      A     M      3.3;
      =     L      0.0;
      A     L      0.0;
      A     I    303.6;
      AN    I    303.7;
      =     M    704.4;
      A     L      0.0;
      AN    I    303.6;
      A     I    303.7;
      =     M    704.5;
NETWORK
TITLE =

      A     M      3.3;
      =     L      0.0;
      A     L      0.0;
      A     I    309.0;
      AN    I    309.1;
      AN    I    307.5;
      =     M    704.6;
      A     L      0.0;
      AN    I    309.0;
      A     I    309.1;
      A     I    307.5;
      =     M    704.7;
NETWORK
TITLE =

      A     M      3.3;
      =     L      0.0;
      A     L      0.0;
      A     I    309.2;
      AN    I    306.6;
      =     M    706.6;
      A     L      0.0;
      AN    I    309.2;
      A     I    306.6;
      =     M    706.7;
NETWORK
TITLE =
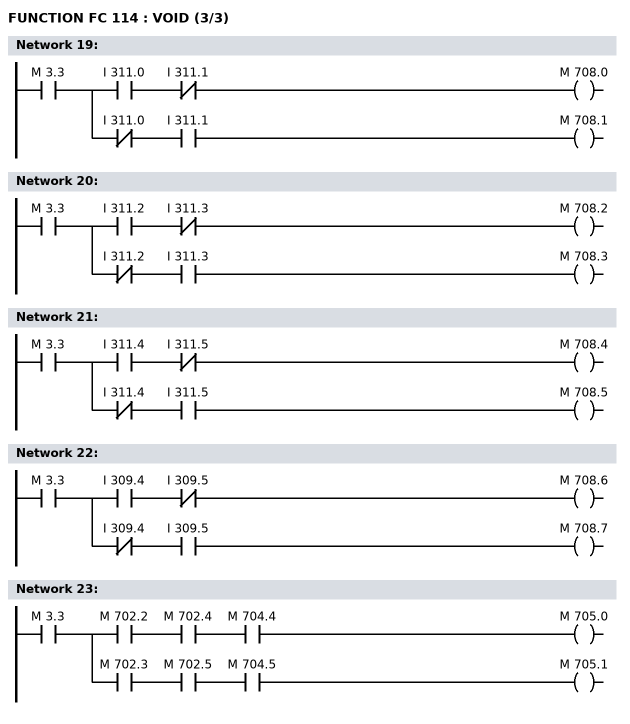

      A     M      3.3;
      =     L      0.0;
      A     L      0.0;
      A     I    311.0;
      AN    I    311.1;
      =     M    708.0;
      A     L      0.0;
      AN    I    311.0;
      A     I    311.1;
      =     M    708.1;
NETWORK
TITLE =

      A     M      3.3;
      =     L      0.0;
      A     L      0.0;
      A     I    311.2;
      AN    I    311.3;
      =     M    708.2;
      A     L      0.0;
      AN    I    311.2;
      A     I    311.3;
      =     M    708.3;
NETWORK
TITLE =

      A     M      3.3;
      =     L      0.0;
      A     L      0.0;
      A     I    311.4;
      AN    I    311.5;
      =     M    708.4;
      A     L      0.0;
      AN    I    311.4;
      A     I    311.5;
      =     M    708.5;
NETWORK
TITLE =

      A     M      3.3;
      =     L      0.0;
      A     L      0.0;
      A     I    309.4;
      AN    I    309.5;
      =     M    708.6;
      A     L      0.0;
      AN    I    309.4;
      A     I    309.5;
      =     M    708.7;
NETWORK
TITLE =

      A     M      3.3;
      =     L      0.0;
      A     L      0.0;
      A     M    702.2;
      A     M    702.4;
      A     M    704.4;
      =     M    705.0;
      A     L      0.0;
      A     M    702.3;
      A     M    702.5;
      A     M    704.5;
      =     M    705.1;
NETWORK
TITLE =

      A     M      3.3;
      =     L      0.0;
      A     L      0.0;
      A     M    702.6;
      A     M    703.0;
      A     M    703.2;
      A     M    703.4;
      A     M    703.6;
      A     M    706.6;
      =     L      0.1;
      A     L      0.1;
      BLD   102;
      =     M    705.2;
      A     L      0.1;
      A     M    704.2;
      A     M    704.6;
      =     M    705.4;
      A     L      0.0;
      A     M    702.7;
      A     M    703.1;
      A     M    703.3;
      A     M    703.5;
      A     M    703.7;
      A     M    706.7;
      =     L      0.1;
      A     L      0.1;
      BLD   102;
      =     M    705.3;
      A     L      0.1;
      A     M    704.3;
      A     M    704.7;
      =     M    705.5;
NETWORK
TITLE =
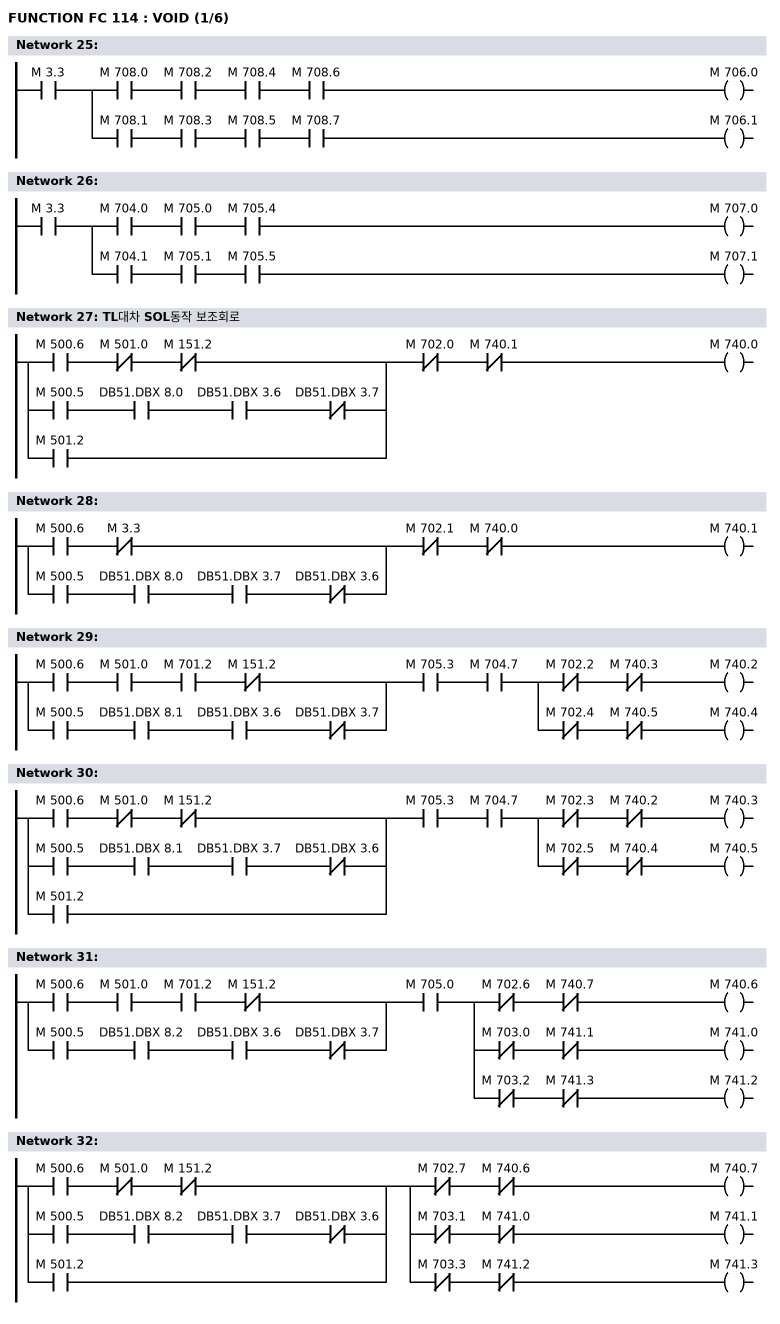

      A     M      3.3;
      =     L      0.0;
      A     L      0.0;
      A     M    708.0;
      A     M    708.2;
      A     M    708.4;
      A     M    708.6;
      =     M    706.0;
      A     L      0.0;
      A     M    708.1;
      A     M    708.3;
      A     M    708.5;
      A     M    708.7;
      =     M    706.1;
NETWORK
TITLE =

      A     M      3.3;
      =     L      0.0;
      A     L      0.0;
      A     M    704.0;
      A     M    705.0;
      A     M    705.4;
      =     M    707.0;
      A     L      0.0;
      A     M    704.1;
      A     M    705.1;
      A     M    705.5;
      =     M    707.1;
NETWORK
TITLE =TL대차 SOL동작 보조회로

      A(    ;
      A     M    500.6;
      AN    M    501.0;
      AN    M    151.2;
      O     ;
      A     M    500.5;
      A     DB51.DBX    8.0;
      A     DB51.DBX    3.6;
      AN    DB51.DBX    3.7;
      O     M    501.2;
      )     ;
      AN    M    702.0;
      AN    M    740.1;
      =     M    740.0;
NETWORK
TITLE =

      A(    ;
      A     M    500.6;
      AN    M      3.3;
      O     ;
      A     M    500.5;
      A     DB51.DBX    8.0;
      A     DB51.DBX    3.7;
      AN    DB51.DBX    3.6;
      )     ;
      AN    M    702.1;
      AN    M    740.0;
      =     M    740.1;
NETWORK
TITLE =

      A(    ;
      A     M    500.6;
      A     M    501.0;
      A     M    701.2;
      AN    M    151.2;
      O     ;
      A     M    500.5;
      A     DB51.DBX    8.1;
      A     DB51.DBX    3.6;
      AN    DB51.DBX    3.7;
      )     ;
      A     M    705.3;
      A     M    704.7;
      =     L      0.0;
      A     L      0.0;
      AN    M    702.2;
      AN    M    740.3;
      =     M    740.2;
      A     L      0.0;
      AN    M    702.4;
      AN    M    740.5;
      =     M    740.4;
NETWORK
TITLE =

      A(    ;
      A     M    500.6;
      AN    M    501.0;
      AN    M    151.2;
      O     ;
      A     M    500.5;
      A     DB51.DBX    8.1;
      A     DB51.DBX    3.7;
      AN    DB51.DBX    3.6;
      O     M    501.2;
      )     ;
      A     M    705.3;
      A     M    704.7;
      =     L      0.0;
      A     L      0.0;
      AN    M    702.3;
      AN    M    740.2;
      =     M    740.3;
      A     L      0.0;
      AN    M    702.5;
      AN    M    740.4;
      =     M    740.5;
NETWORK
TITLE =

      A(    ;
      A     M    500.6;
      A     M    501.0;
      A     M    701.2;
      AN    M    151.2;
      O     ;
      A     M    500.5;
      A     DB51.DBX    8.2;
      A     DB51.DBX    3.6;
      AN    DB51.DBX    3.7;
      )     ;
      A     M    705.0;
      =     L      0.0;
      A     L      0.0;
      AN    M    702.6;
      AN    M    740.7;
      =     M    740.6;
      A     L      0.0;
      AN    M    703.0;
      AN    M    741.1;
      =     M    741.0;
      A     L      0.0;
      AN    M    703.2;
      AN    M    741.3;
      =     M    741.2;
NETWORK
TITLE =

      A     M    500.6;
      AN    M    501.0;
      AN    M    151.2;
      O     ;
      A     M    500.5;
      A     DB51.DBX    8.2;
      A     DB51.DBX    3.7;
      AN    DB51.DBX    3.6;
      O     M    501.2;
      =     L      0.0;
      A     L      0.0;
      AN    M    702.7;
      AN    M    740.6;
      =     M    740.7;
      A     L      0.0;
      AN    M    703.1;
      AN    M    741.0;
      =     M    741.1;
      A     L      0.0;
      AN    M    703.3;
      AN    M    741.2;
      =     M    741.3;
NETWORK
TITLE =
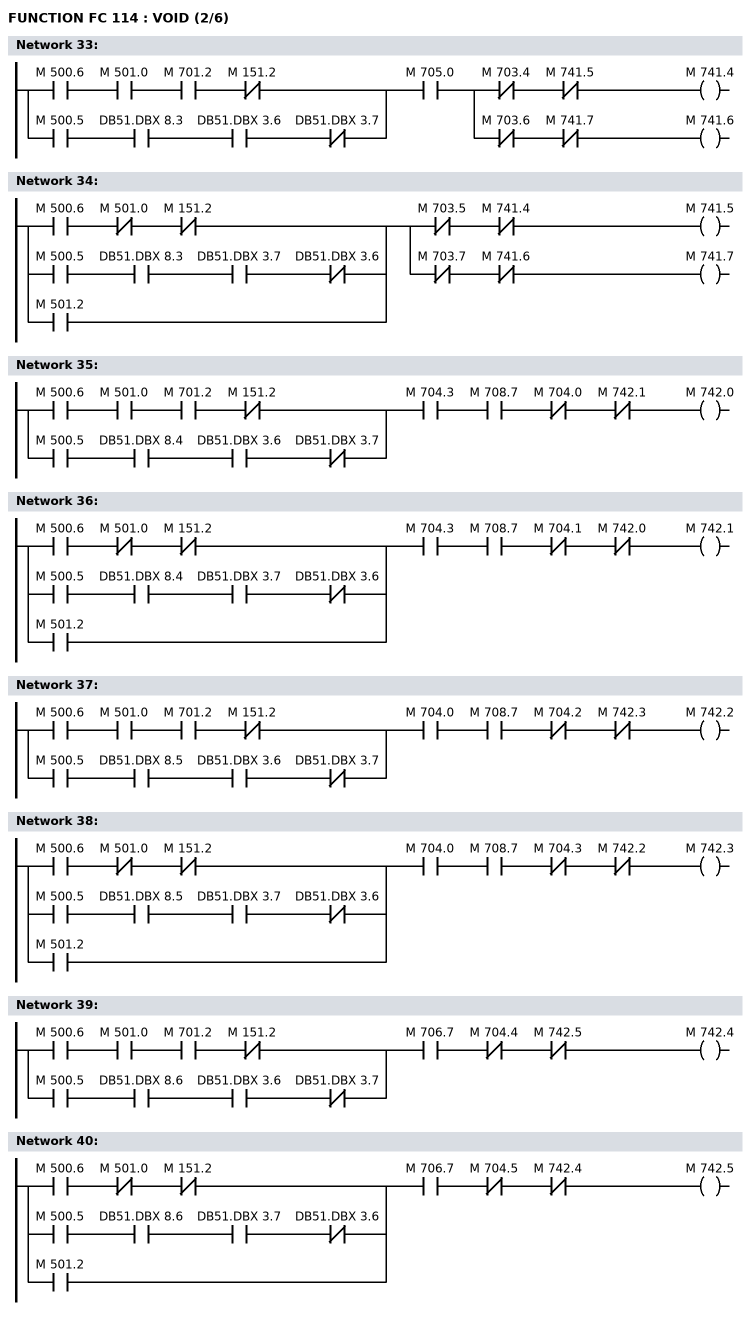

      A(    ;
      A     M    500.6;
      A     M    501.0;
      A     M    701.2;
      AN    M    151.2;
      O     ;
      A     M    500.5;
      A     DB51.DBX    8.3;
      A     DB51.DBX    3.6;
      AN    DB51.DBX    3.7;
      )     ;
      A     M    705.0;
      =     L      0.0;
      A     L      0.0;
      AN    M    703.4;
      AN    M    741.5;
      =     M    741.4;
      A     L      0.0;
      AN    M    703.6;
      AN    M    741.7;
      =     M    741.6;
NETWORK
TITLE =

      A     M    500.6;
      AN    M    501.0;
      AN    M    151.2;
      O     ;
      A     M    500.5;
      A     DB51.DBX    8.3;
      A     DB51.DBX    3.7;
      AN    DB51.DBX    3.6;
      O     M    501.2;
      =     L      0.0;
      A     L      0.0;
      AN    M    703.5;
      AN    M    741.4;
      =     M    741.5;
      A     L      0.0;
      AN    M    703.7;
      AN    M    741.6;
      =     M    741.7;
NETWORK
TITLE =

      A(    ;
      A     M    500.6;
      A     M    501.0;
      A     M    701.2;
      AN    M    151.2;
      O     ;
      A     M    500.5;
      A     DB51.DBX    8.4;
      A     DB51.DBX    3.6;
      AN    DB51.DBX    3.7;
      )     ;
      A     M    704.3;
      A     M    708.7;
      AN    M    704.0;
      AN    M    742.1;
      =     M    742.0;
NETWORK
TITLE =

      A(    ;
      A     M    500.6;
      AN    M    501.0;
      AN    M    151.2;
      O     ;
      A     M    500.5;
      A     DB51.DBX    8.4;
      A     DB51.DBX    3.7;
      AN    DB51.DBX    3.6;
      O     M    501.2;
      )     ;
      A     M    704.3;
      A     M    708.7;
      AN    M    704.1;
      AN    M    742.0;
      =     M    742.1;
NETWORK
TITLE =

      A(    ;
      A     M    500.6;
      A     M    501.0;
      A     M    701.2;
      AN    M    151.2;
      O     ;
      A     M    500.5;
      A     DB51.DBX    8.5;
      A     DB51.DBX    3.6;
      AN    DB51.DBX    3.7;
      )     ;
      A     M    704.0;
      A     M    708.7;
      AN    M    704.2;
      AN    M    742.3;
      =     M    742.2;
NETWORK
TITLE =

      A(    ;
      A     M    500.6;
      AN    M    501.0;
      AN    M    151.2;
      O     ;
      A     M    500.5;
      A     DB51.DBX    8.5;
      A     DB51.DBX    3.7;
      AN    DB51.DBX    3.6;
      O     M    501.2;
      )     ;
      A     M    704.0;
      A     M    708.7;
      AN    M    704.3;
      AN    M    742.2;
      =     M    742.3;
NETWORK
TITLE =

      A(    ;
      A     M    500.6;
      A     M    501.0;
      A     M    701.2;
      AN    M    151.2;
      O     ;
      A     M    500.5;
      A     DB51.DBX    8.6;
      A     DB51.DBX    3.6;
      AN    DB51.DBX    3.7;
      )     ;
      A     M    706.7;
      AN    M    704.4;
      AN    M    742.5;
      =     M    742.4;
NETWORK
TITLE =

      A(    ;
      A     M    500.6;
      AN    M    501.0;
      AN    M    151.2;
      O     ;
      A     M    500.5;
      A     DB51.DBX    8.6;
      A     DB51.DBX    3.7;
      AN    DB51.DBX    3.6;
      O     M    501.2;
      )     ;
      A     M    706.7;
      AN    M    704.5;
      AN    M    742.4;
      =     M    742.5;
NETWORK
TITLE =
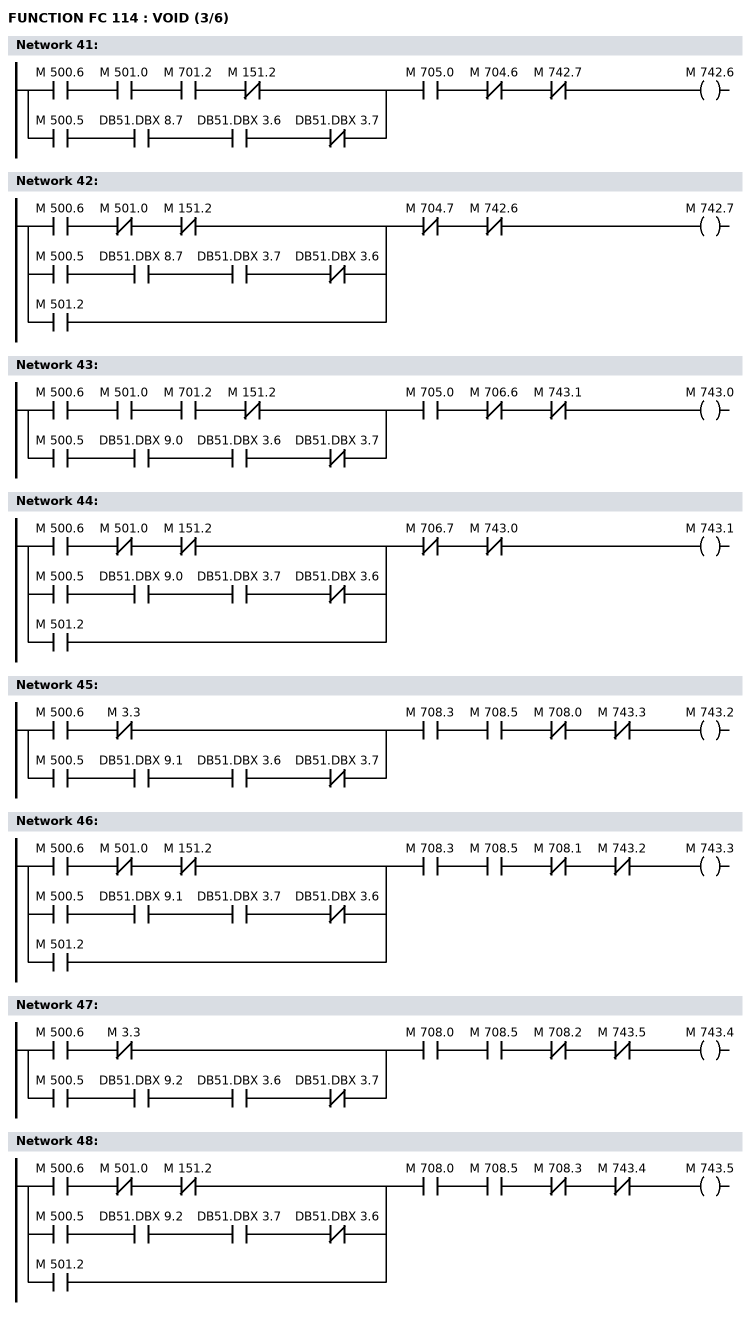

      A(    ;
      A     M    500.6;
      A     M    501.0;
      A     M    701.2;
      AN    M    151.2;
      O     ;
      A     M    500.5;
      A     DB51.DBX    8.7;
      A     DB51.DBX    3.6;
      AN    DB51.DBX    3.7;
      )     ;
      A     M    705.0;
      AN    M    704.6;
      AN    M    742.7;
      =     M    742.6;
NETWORK
TITLE =

      A(    ;
      A     M    500.6;
      AN    M    501.0;
      AN    M    151.2;
      O     ;
      A     M    500.5;
      A     DB51.DBX    8.7;
      A     DB51.DBX    3.7;
      AN    DB51.DBX    3.6;
      O     M    501.2;
      )     ;
      AN    M    704.7;
      AN    M    742.6;
      =     M    742.7;
NETWORK
TITLE =

      A(    ;
      A     M    500.6;
      A     M    501.0;
      A     M    701.2;
      AN    M    151.2;
      O     ;
      A     M    500.5;
      A     DB51.DBX    9.0;
      A     DB51.DBX    3.6;
      AN    DB51.DBX    3.7;
      )     ;
      A     M    705.0;
      AN    M    706.6;
      AN    M    743.1;
      =     M    743.0;
NETWORK
TITLE =

      A(    ;
      A     M    500.6;
      AN    M    501.0;
      AN    M    151.2;
      O     ;
      A     M    500.5;
      A     DB51.DBX    9.0;
      A     DB51.DBX    3.7;
      AN    DB51.DBX    3.6;
      O     M    501.2;
      )     ;
      AN    M    706.7;
      AN    M    743.0;
      =     M    743.1;
NETWORK
TITLE =

      A(    ;
      A     M    500.6;
      AN    M      3.3;
      O     ;
      A     M    500.5;
      A     DB51.DBX    9.1;
      A     DB51.DBX    3.6;
      AN    DB51.DBX    3.7;
      )     ;
      A     M    708.3;
      A     M    708.5;
      AN    M    708.0;
      AN    M    743.3;
      =     M    743.2;
NETWORK
TITLE =

      A(    ;
      A     M    500.6;
      AN    M    501.0;
      AN    M    151.2;
      O     ;
      A     M    500.5;
      A     DB51.DBX    9.1;
      A     DB51.DBX    3.7;
      AN    DB51.DBX    3.6;
      O     M    501.2;
      )     ;
      A     M    708.3;
      A     M    708.5;
      AN    M    708.1;
      AN    M    743.2;
      =     M    743.3;
NETWORK
TITLE =

      A(    ;
      A     M    500.6;
      AN    M      3.3;
      O     ;
      A     M    500.5;
      A     DB51.DBX    9.2;
      A     DB51.DBX    3.6;
      AN    DB51.DBX    3.7;
      )     ;
      A     M    708.0;
      A     M    708.5;
      AN    M    708.2;
      AN    M    743.5;
      =     M    743.4;
NETWORK
TITLE =

      A(    ;
      A     M    500.6;
      AN    M    501.0;
      AN    M    151.2;
      O     ;
      A     M    500.5;
      A     DB51.DBX    9.2;
      A     DB51.DBX    3.7;
      AN    DB51.DBX    3.6;
      O     M    501.2;
      )     ;
      A     M    708.0;
      A     M    708.5;
      AN    M    708.3;
      AN    M    743.4;
      =     M    743.5;
NETWORK
TITLE =
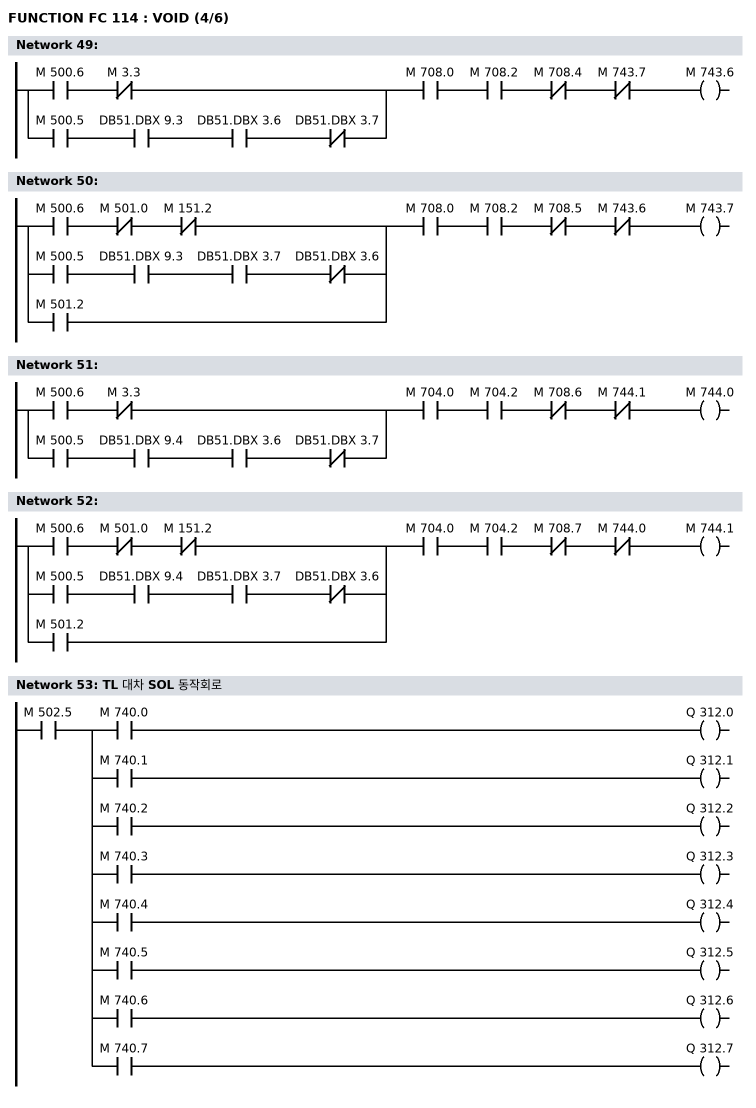

      A(    ;
      A     M    500.6;
      AN    M      3.3;
      O     ;
      A     M    500.5;
      A     DB51.DBX    9.3;
      A     DB51.DBX    3.6;
      AN    DB51.DBX    3.7;
      )     ;
      A     M    708.0;
      A     M    708.2;
      AN    M    708.4;
      AN    M    743.7;
      =     M    743.6;
NETWORK
TITLE =

      A(    ;
      A     M    500.6;
      AN    M    501.0;
      AN    M    151.2;
      O     ;
      A     M    500.5;
      A     DB51.DBX    9.3;
      A     DB51.DBX    3.7;
      AN    DB51.DBX    3.6;
      O     M    501.2;
      )     ;
      A     M    708.0;
      A     M    708.2;
      AN    M    708.5;
      AN    M    743.6;
      =     M    743.7;
NETWORK
TITLE =

      A(    ;
      A     M    500.6;
      AN    M      3.3;
      O     ;
      A     M    500.5;
      A     DB51.DBX    9.4;
      A     DB51.DBX    3.6;
      AN    DB51.DBX    3.7;
      )     ;
      A     M    704.0;
      A     M    704.2;
      AN    M    708.6;
      AN    M    744.1;
      =     M    744.0;
NETWORK
TITLE =

      A(    ;
      A     M    500.6;
      AN    M    501.0;
      AN    M    151.2;
      O     ;
      A     M    500.5;
      A     DB51.DBX    9.4;
      A     DB51.DBX    3.7;
      AN    DB51.DBX    3.6;
      O     M    501.2;
      )     ;
      A     M    704.0;
      A     M    704.2;
      AN    M    708.7;
      AN    M    744.0;
      =     M    744.1;
NETWORK
TITLE =TL 대차 SOL 동작회로

      A     M    502.5;
      =     L      0.0;
      A     L      0.0;
      A     M    740.0;
      =     Q    312.0;
      A     L      0.0;
      A     M    740.1;
      =     Q    312.1;
      A     L      0.0;
      A     M    740.2;
      =     Q    312.2;
      A     L      0.0;
      A     M    740.3;
      =     Q    312.3;
      A     L      0.0;
      A     M    740.4;
      =     Q    312.4;
      A     L      0.0;
      A     M    740.5;
      =     Q    312.5;
      A     L      0.0;
      A     M    740.6;
      =     Q    312.6;
      A     L      0.0;
      A     M    740.7;
      =     Q    312.7;
NETWORK
TITLE =
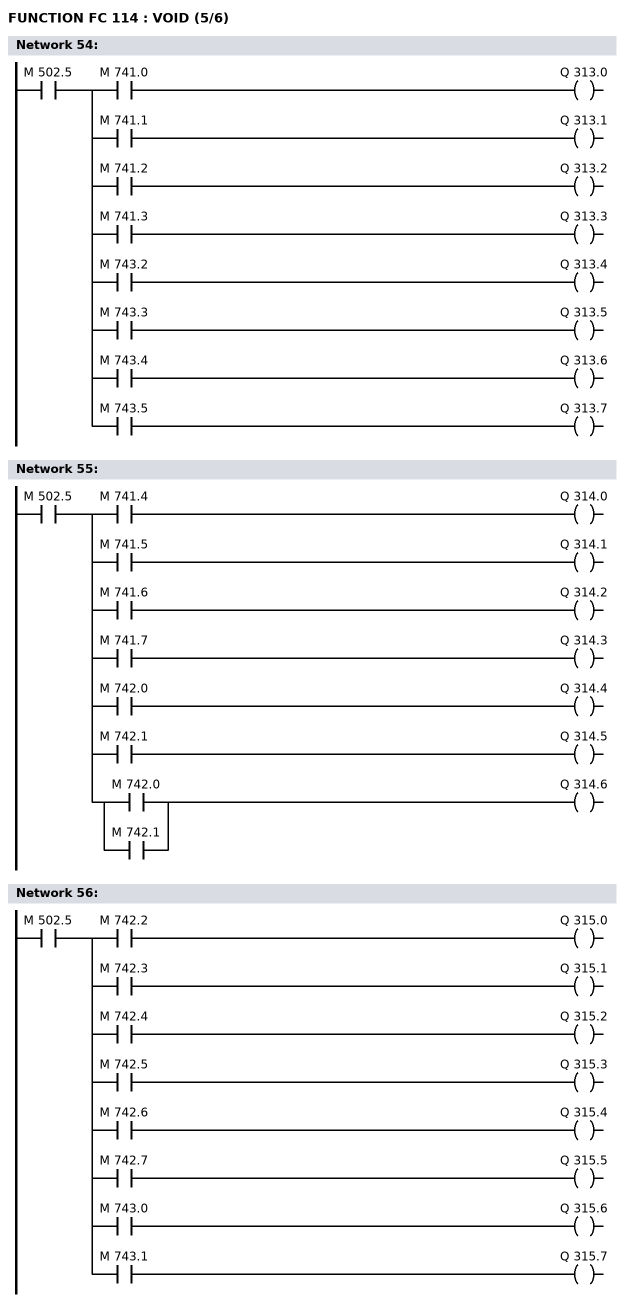

      A     M    502.5;
      =     L      0.0;
      A     L      0.0;
      A     M    741.0;
      =     Q    313.0;
      A     L      0.0;
      A     M    741.1;
      =     Q    313.1;
      A     L      0.0;
      A     M    741.2;
      =     Q    313.2;
      A     L      0.0;
      A     M    741.3;
      =     Q    313.3;
      A     L      0.0;
      A     M    743.2;
      =     Q    313.4;
      A     L      0.0;
      A     M    743.3;
      =     Q    313.5;
      A     L      0.0;
      A     M    743.4;
      =     Q    313.6;
      A     L      0.0;
      A     M    743.5;
      =     Q    313.7;
NETWORK
TITLE =

      A     M    502.5;
      =     L      0.0;
      A     L      0.0;
      A     M    741.4;
      =     Q    314.0;
      A     L      0.0;
      A     M    741.5;
      =     Q    314.1;
      A     L      0.0;
      A     M    741.6;
      =     Q    314.2;
      A     L      0.0;
      A     M    741.7;
      =     Q    314.3;
      A     L      0.0;
      A     M    742.0;
      =     Q    314.4;
      A     L      0.0;
      A     M    742.1;
      =     Q    314.5;
      A     L      0.0;
      A(    ;
      O     M    742.0;
      O     M    742.1;
      )     ;
      =     Q    314.6;
NETWORK
TITLE =

      A     M    502.5;
      =     L      0.0;
      A     L      0.0;
      A     M    742.2;
      =     Q    315.0;
      A     L      0.0;
      A     M    742.3;
      =     Q    315.1;
      A     L      0.0;
      A     M    742.4;
      =     Q    315.2;
      A     L      0.0;
      A     M    742.5;
      =     Q    315.3;
      A     L      0.0;
      A     M    742.6;
      =     Q    315.4;
      A     L      0.0;
      A     M    742.7;
      =     Q    315.5;
      A     L      0.0;
      A     M    743.0;
      =     Q    315.6;
      A     L      0.0;
      A     M    743.1;
      =     Q    315.7;
NETWORK
TITLE =
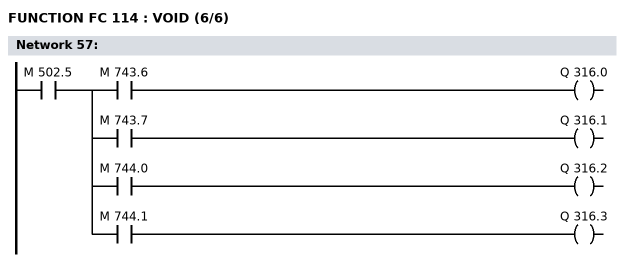

      A     M    502.5;
      =     L      0.0;
      A     L      0.0;
      A     M    743.6;
      =     Q    316.0;
      A     L      0.0;
      A     M    743.7;
      =     Q    316.1;
      A     L      0.0;
      A     M    744.0;
      =     Q    316.2;
      A     L      0.0;
      A     M    744.1;
      =     Q    316.3;
END_FUNCTION

FUNCTION FC 115 : VOID
TITLE =
VERSION : 0.1

BEGIN
NETWORK
TITLE =
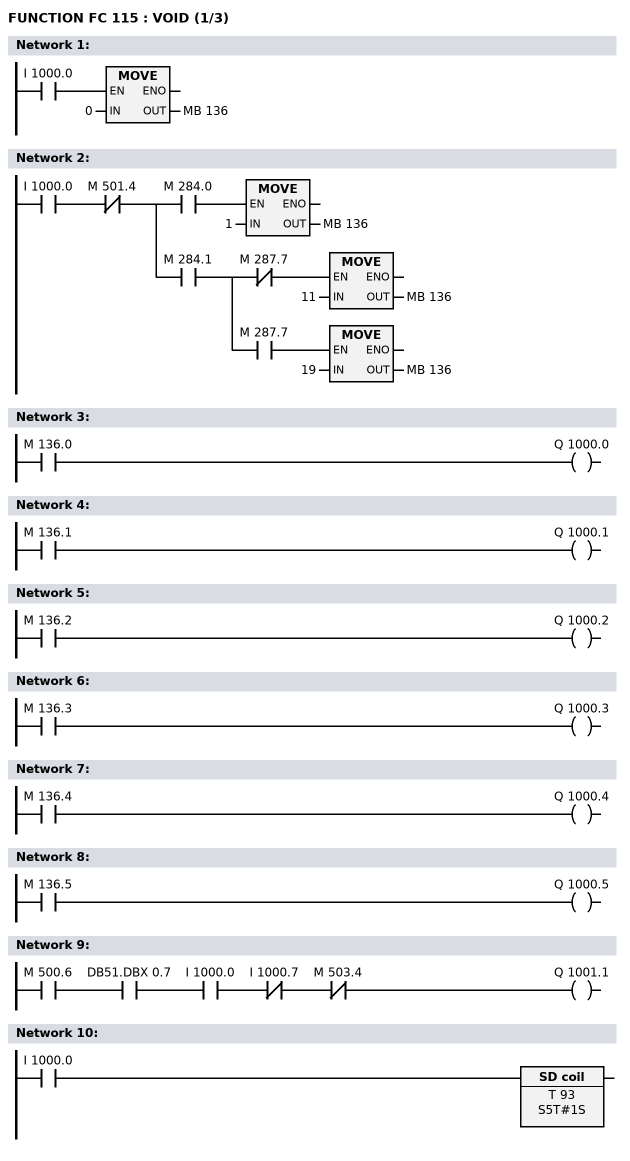

      A     I   1000.0;
      JNB   _001;
      L     0;
      T     MB   136;
_001: NOP   0;
NETWORK
TITLE =

      A     I   1000.0;
      AN    M    501.4;
      =     L      0.0;
      A     L      0.0;
      A     M    284.0;
      JNB   _002;
      L     1;
      T     MB   136;
_002: NOP   0;
      A     L      0.0;
      A     M    284.1;
      =     L      0.1;
      A     L      0.1;
      AN    M    287.7;
      JNB   _003;
      L     11;
      T     MB   136;
_003: NOP   0;
      A     L      0.1;
      A     M    287.7;
      JNB   _004;
      L     19;
      T     MB   136;
_004: NOP   0;
NETWORK
TITLE =

      A     M    136.0;
      =     Q   1000.0;
NETWORK
TITLE =

      A     M    136.1;
      =     Q   1000.1;
NETWORK
TITLE =

      A     M    136.2;
      =     Q   1000.2;
NETWORK
TITLE =

      A     M    136.3;
      =     Q   1000.3;
NETWORK
TITLE =

      A     M    136.4;
      =     Q   1000.4;
NETWORK
TITLE =

      A     M    136.5;
      =     Q   1000.5;
NETWORK
TITLE =

      A     M    500.6;
      A     DB51.DBX    0.7;
      A     I   1000.0;
      AN    I   1000.7;
      AN    M    503.4;
      =     Q   1001.1;
NETWORK
TITLE =

      A     I   1000.0;
      L     S5T#1S;
      SD    T     93;
NETWORK
TITLE =
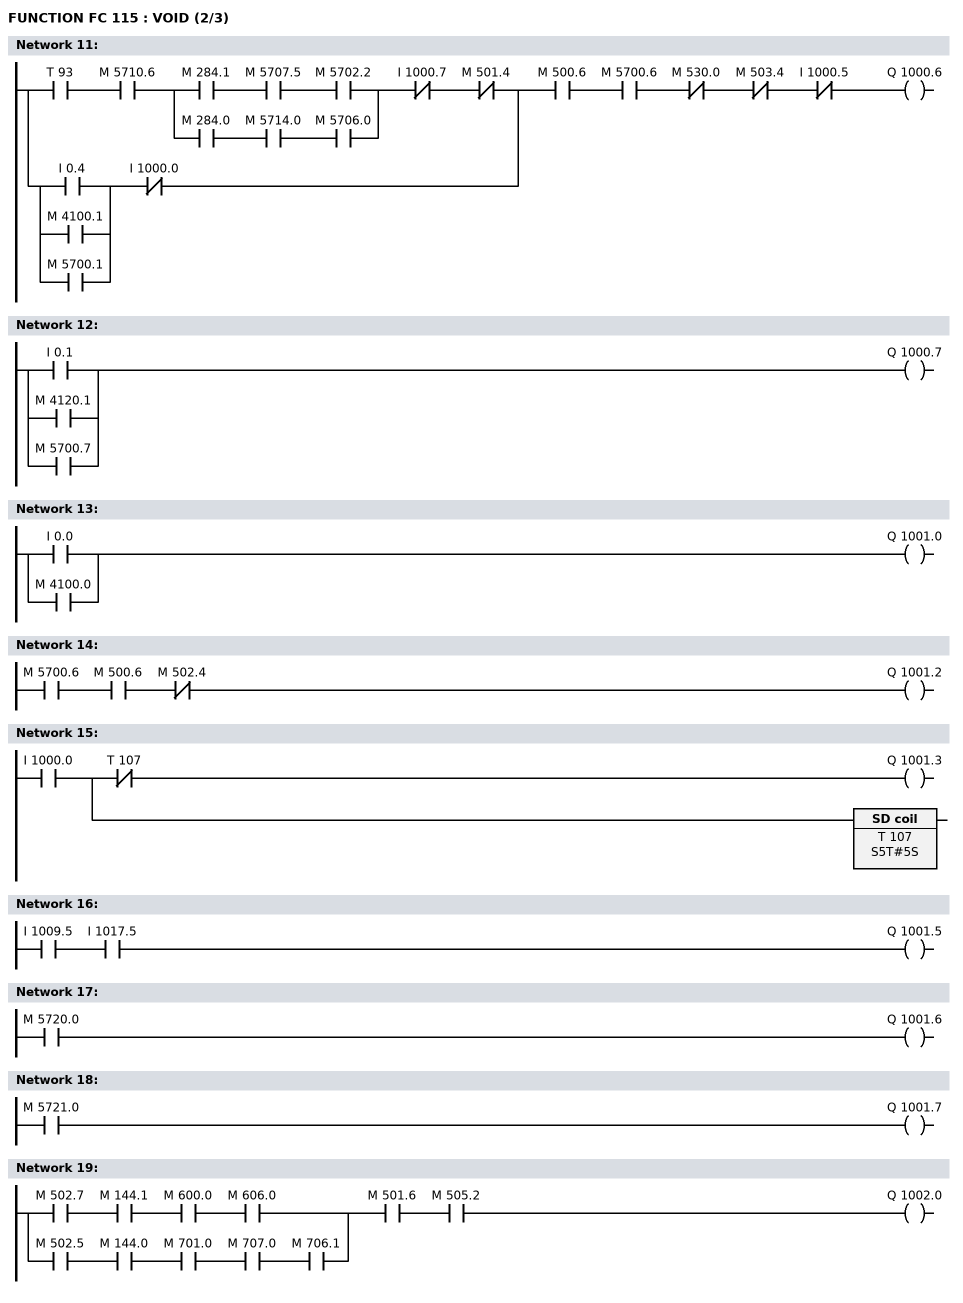

      A(    ;
      A     T     93;
      A     M   5710.6;
      A(    ;
      A     M    284.1;
      A     M   5707.5;
      A     M   5702.2;
      O     ;
      A     M    284.0;
      A     M   5714.0;
      A     M   5706.0;
      )     ;
      AN    I   1000.7;
      AN    M    501.4;
      O     ;
      A(    ;
      O     I      0.4;
      O     M   4100.1;
      O     M   5700.1;
      )     ;
      AN    I   1000.0;
      )     ;
      A     M    500.6;
      A     M   5700.6;
      AN    M    530.0;
      AN    M    503.4;
      AN    I   1000.5;
      =     Q   1000.6;
NETWORK
TITLE =

      O     I      0.1;
      O     M   4120.1;
      O     M   5700.7;
      =     Q   1000.7;
NETWORK
TITLE =

      O     I      0.0;
      O     M   4100.0;
      =     Q   1001.0;
NETWORK
TITLE =

      A     M   5700.6;
      A     M    500.6;
      AN    M    502.4;
      =     Q   1001.2;
NETWORK
TITLE =

      A     I   1000.0;
      =     L      0.0;
      A     L      0.0;
      AN    T    107;
      =     Q   1001.3;
      A     L      0.0;
      BLD   102;
      L     S5T#5S;
      SD    T    107;
NETWORK
TITLE =

      A     I   1009.5;
      A     I   1017.5;
      =     Q   1001.5;
NETWORK
TITLE =

      A     M   5720.0;
      =     Q   1001.6;
NETWORK
TITLE =

      A     M   5721.0;
      =     Q   1001.7;
NETWORK
TITLE =

      A(    ;
      A     M    502.7;
      A     M    144.1;
      A     M    600.0;
      A     M    606.0;
      O     ;
      A     M    502.5;
      A     M    144.0;
      A     M    701.0;
      A     M    707.0;
      A     M    706.1;
      )     ;
      A     M    501.6;
      A     M    505.2;
      =     Q   1002.0;
NETWORK
TITLE =
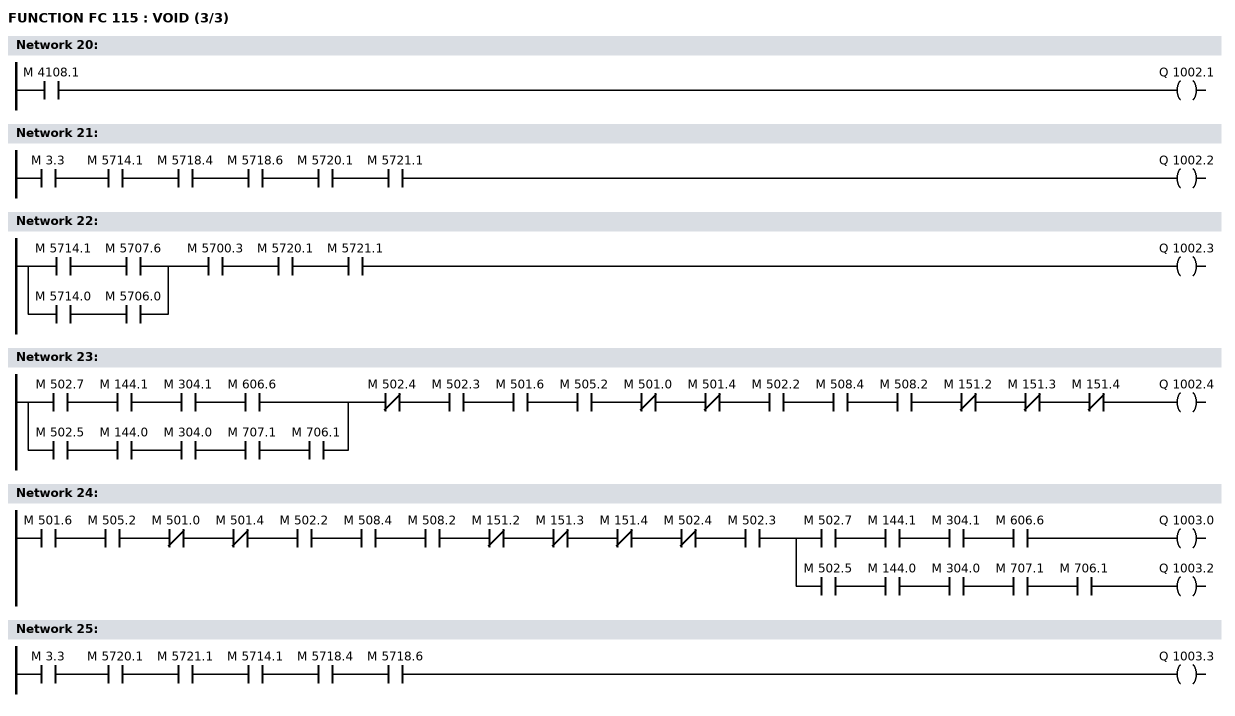

      A     M   4108.1;
      =     Q   1002.1;
NETWORK
TITLE =

      A     M      3.3;
      A     M   5714.1;
      A     M   5718.4;
      A     M   5718.6;
      A     M   5720.1;
      A     M   5721.1;
      =     Q   1002.2;
NETWORK
TITLE =

      A(    ;
      A     M   5714.1;
      A     M   5707.6;
      O     ;
      A     M   5714.0;
      A     M   5706.0;
      )     ;
      A     M   5700.3;
      A     M   5720.1;
      A     M   5721.1;
      =     Q   1002.3;
NETWORK
TITLE =

      A(    ;
      A     M    502.7;
      A     M    144.1;
      A     M    304.1;
      A     M    606.6;
      O     ;
      A     M    502.5;
      A     M    144.0;
      A     M    304.0;
      A     M    707.1;
      A     M    706.1;
      )     ;
      AN    M    502.4;
      A     M    502.3;
      A     M    501.6;
      A     M    505.2;
      AN    M    501.0;
      AN    M    501.4;
      A     M    502.2;
      A     M    508.4;
      A     M    508.2;
      AN    M    151.2;
      AN    M    151.3;
      AN    M    151.4;
      =     Q   1002.4;
NETWORK
TITLE =

      A     M    501.6;
      A     M    505.2;
      AN    M    501.0;
      AN    M    501.4;
      A     M    502.2;
      A     M    508.4;
      A     M    508.2;
      AN    M    151.2;
      AN    M    151.3;
      AN    M    151.4;
      AN    M    502.4;
      A     M    502.3;
      =     L      0.0;
      A     L      0.0;
      A     M    502.7;
      A     M    144.1;
      A     M    304.1;
      A     M    606.6;
      =     Q   1003.0;
      A     L      0.0;
      A     M    502.5;
      A     M    144.0;
      A     M    304.0;
      A     M    707.1;
      A     M    706.1;
      =     Q   1003.2;
NETWORK
TITLE =

      A     M      3.3;
      A     M   5720.1;
      A     M   5721.1;
      A     M   5714.1;
      A     M   5718.4;
      A     M   5718.6;
      =     Q   1003.3;
END_FUNCTION

FUNCTION FC 116 : VOID
TITLE =
VERSION : 0.1

BEGIN
NETWORK
TITLE =
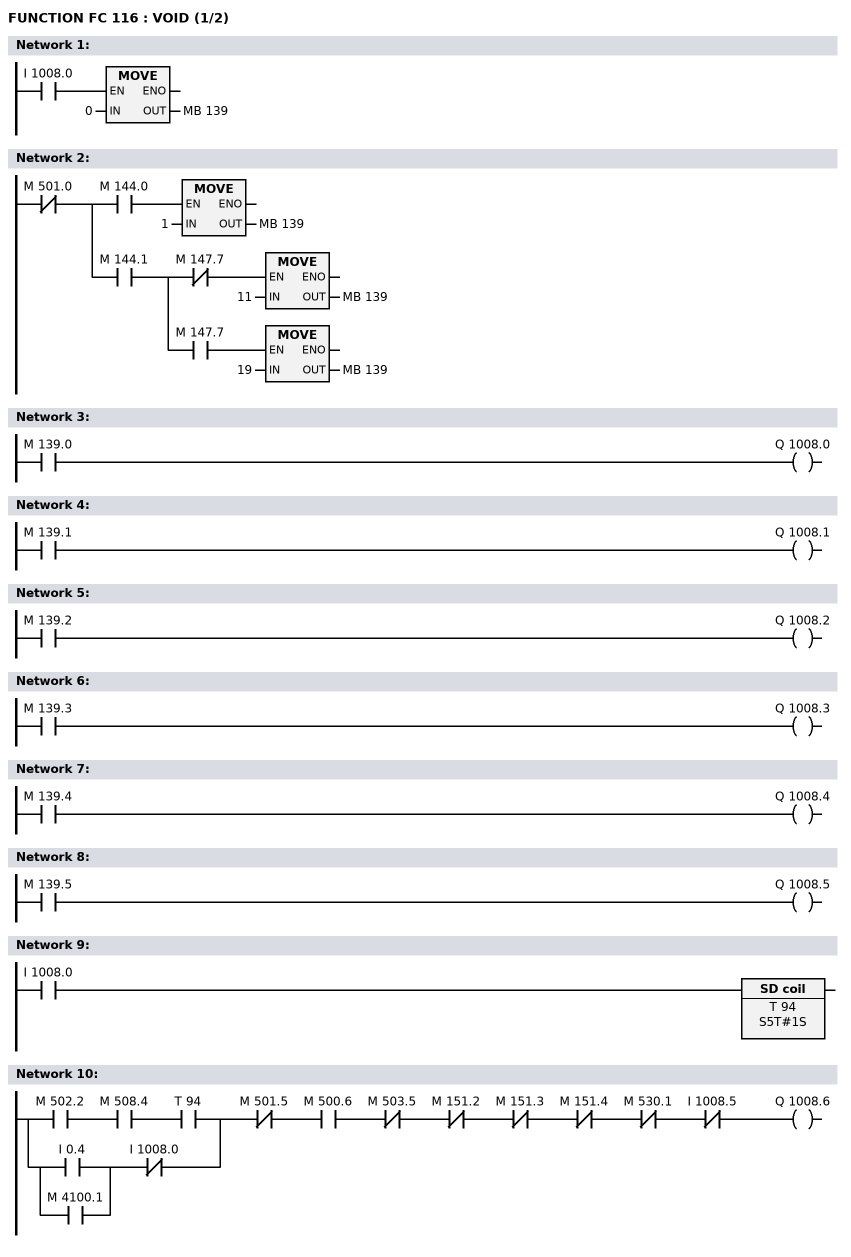

      A     I   1008.0;
      JNB   _001;
      L     0;
      T     MB   139;
_001: NOP   0;
NETWORK
TITLE =

      AN    M    501.0;
      =     L      0.0;
      A     L      0.0;
      A     M    144.0;
      JNB   _002;
      L     1;
      T     MB   139;
_002: NOP   0;
      A     L      0.0;
      A     M    144.1;
      =     L      0.1;
      A     L      0.1;
      AN    M    147.7;
      JNB   _003;
      L     11;
      T     MB   139;
_003: NOP   0;
      A     L      0.1;
      A     M    147.7;
      JNB   _004;
      L     19;
      T     MB   139;
_004: NOP   0;
NETWORK
TITLE =

      A     M    139.0;
      =     Q   1008.0;
NETWORK
TITLE =

      A     M    139.1;
      =     Q   1008.1;
NETWORK
TITLE =

      A     M    139.2;
      =     Q   1008.2;
NETWORK
TITLE =

      A     M    139.3;
      =     Q   1008.3;
NETWORK
TITLE =

      A     M    139.4;
      =     Q   1008.4;
NETWORK
TITLE =

      A     M    139.5;
      =     Q   1008.5;
NETWORK
TITLE =

      A     I   1008.0;
      L     S5T#1S;
      SD    T     94;
NETWORK
TITLE =

      A(    ;
      A     M    502.2;
      A     M    508.4;
      A     T     94;
      O     ;
      A(    ;
      O     I      0.4;
      O     M   4100.1;
      )     ;
      AN    I   1008.0;
      )     ;
      AN    M    501.5;
      A     M    500.6;
      AN    M    503.5;
      AN    M    151.2;
      AN    M    151.3;
      AN    M    151.4;
      AN    M    530.1;
      AN    I   1008.5;
      =     Q   1008.6;
NETWORK
TITLE =
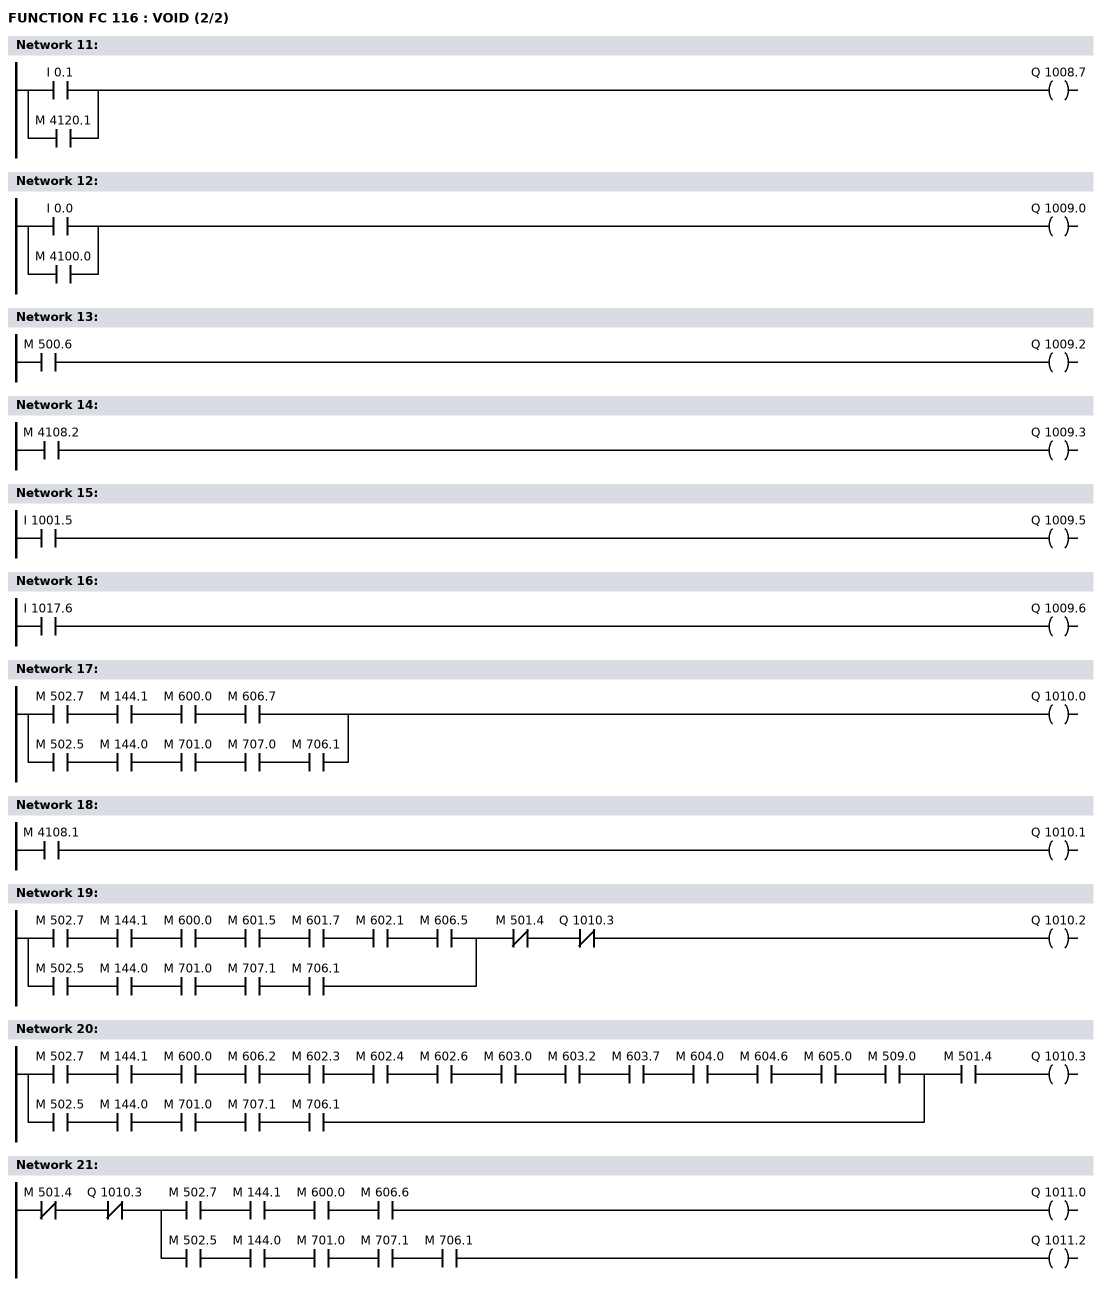

      O     I      0.1;
      O     M   4120.1;
      =     Q   1008.7;
NETWORK
TITLE =

      O     I      0.0;
      O     M   4100.0;
      =     Q   1009.0;
NETWORK
TITLE =

      A     M    500.6;
      =     Q   1009.2;
NETWORK
TITLE =

      A     M   4108.2;
      =     Q   1009.3;
NETWORK
TITLE =

      A     I   1001.5;
      =     Q   1009.5;
NETWORK
TITLE =

      A     I   1017.6;
      =     Q   1009.6;
NETWORK
TITLE =

      A     M    502.7;
      A     M    144.1;
      A     M    600.0;
      A     M    606.7;
      O     ;
      A     M    502.5;
      A     M    144.0;
      A     M    701.0;
      A     M    707.0;
      A     M    706.1;
      =     Q   1010.0;
NETWORK
TITLE =

      A     M   4108.1;
      =     Q   1010.1;
NETWORK
TITLE =

      A(    ;
      A     M    502.7;
      A     M    144.1;
      A     M    600.0;
      A     M    601.5;
      A     M    601.7;
      A     M    602.1;
      A     M    606.5;
      O     ;
      A     M    502.5;
      A     M    144.0;
      A     M    701.0;
      A     M    707.1;
      A     M    706.1;
      )     ;
      AN    M    501.4;
      AN    Q   1010.3;
      =     Q   1010.2;
NETWORK
TITLE =

      A(    ;
      A     M    502.7;
      A     M    144.1;
      A     M    600.0;
      A     M    606.2;
      A     M    602.3;
      A     M    602.4;
      A     M    602.6;
      A     M    603.0;
      A     M    603.2;
      A     M    603.7;
      A     M    604.0;
      A     M    604.6;
      A     M    605.0;
      A     M    509.0;
      O     ;
      A     M    502.5;
      A     M    144.0;
      A     M    701.0;
      A     M    707.1;
      A     M    706.1;
      )     ;
      A     M    501.4;
      =     Q   1010.3;
NETWORK
TITLE =

      AN    M    501.4;
      AN    Q   1010.3;
      =     L      0.0;
      A     L      0.0;
      A     M    502.7;
      A     M    144.1;
      A     M    600.0;
      A     M    606.6;
      =     Q   1011.0;
      A     L      0.0;
      A     M    502.5;
      A     M    144.0;
      A     M    701.0;
      A     M    707.1;
      A     M    706.1;
      =     Q   1011.2;
END_FUNCTION

FUNCTION FC 117 : VOID
TITLE =
VERSION : 0.1

BEGIN
NETWORK
TITLE =
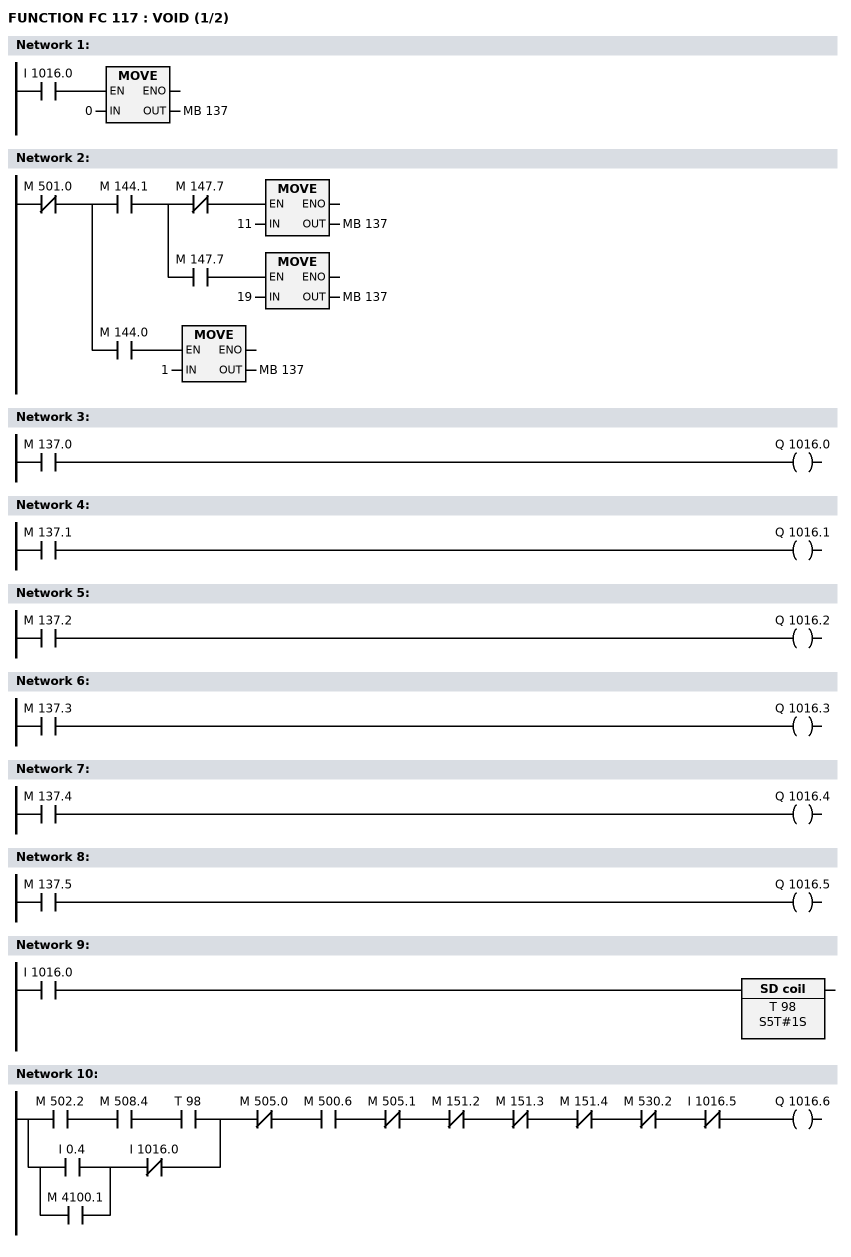

      A     I   1016.0;
      JNB   _001;
      L     0;
      T     MB   137;
_001: NOP   0;
NETWORK
TITLE =

      AN    M    501.0;
      =     L      0.0;
      A     L      0.0;
      A     M    144.1;
      =     L      0.1;
      A     L      0.1;
      AN    M    147.7;
      JNB   _002;
      L     11;
      T     MB   137;
_002: NOP   0;
      A     L      0.1;
      A     M    147.7;
      JNB   _003;
      L     19;
      T     MB   137;
_003: NOP   0;
      A     L      0.0;
      A     M    144.0;
      JNB   _004;
      L     1;
      T     MB   137;
_004: NOP   0;
NETWORK
TITLE =

      A     M    137.0;
      =     Q   1016.0;
NETWORK
TITLE =

      A     M    137.1;
      =     Q   1016.1;
NETWORK
TITLE =

      A     M    137.2;
      =     Q   1016.2;
NETWORK
TITLE =

      A     M    137.3;
      =     Q   1016.3;
NETWORK
TITLE =

      A     M    137.4;
      =     Q   1016.4;
NETWORK
TITLE =

      A     M    137.5;
      =     Q   1016.5;
NETWORK
TITLE =

      A     I   1016.0;
      L     S5T#1S;
      SD    T     98;
NETWORK
TITLE =

      A(    ;
      A     M    502.2;
      A     M    508.4;
      A     T     98;
      O     ;
      A(    ;
      O     I      0.4;
      O     M   4100.1;
      )     ;
      AN    I   1016.0;
      )     ;
      AN    M    505.0;
      A     M    500.6;
      AN    M    505.1;
      AN    M    151.2;
      AN    M    151.3;
      AN    M    151.4;
      AN    M    530.2;
      AN    I   1016.5;
      =     Q   1016.6;
NETWORK
TITLE =
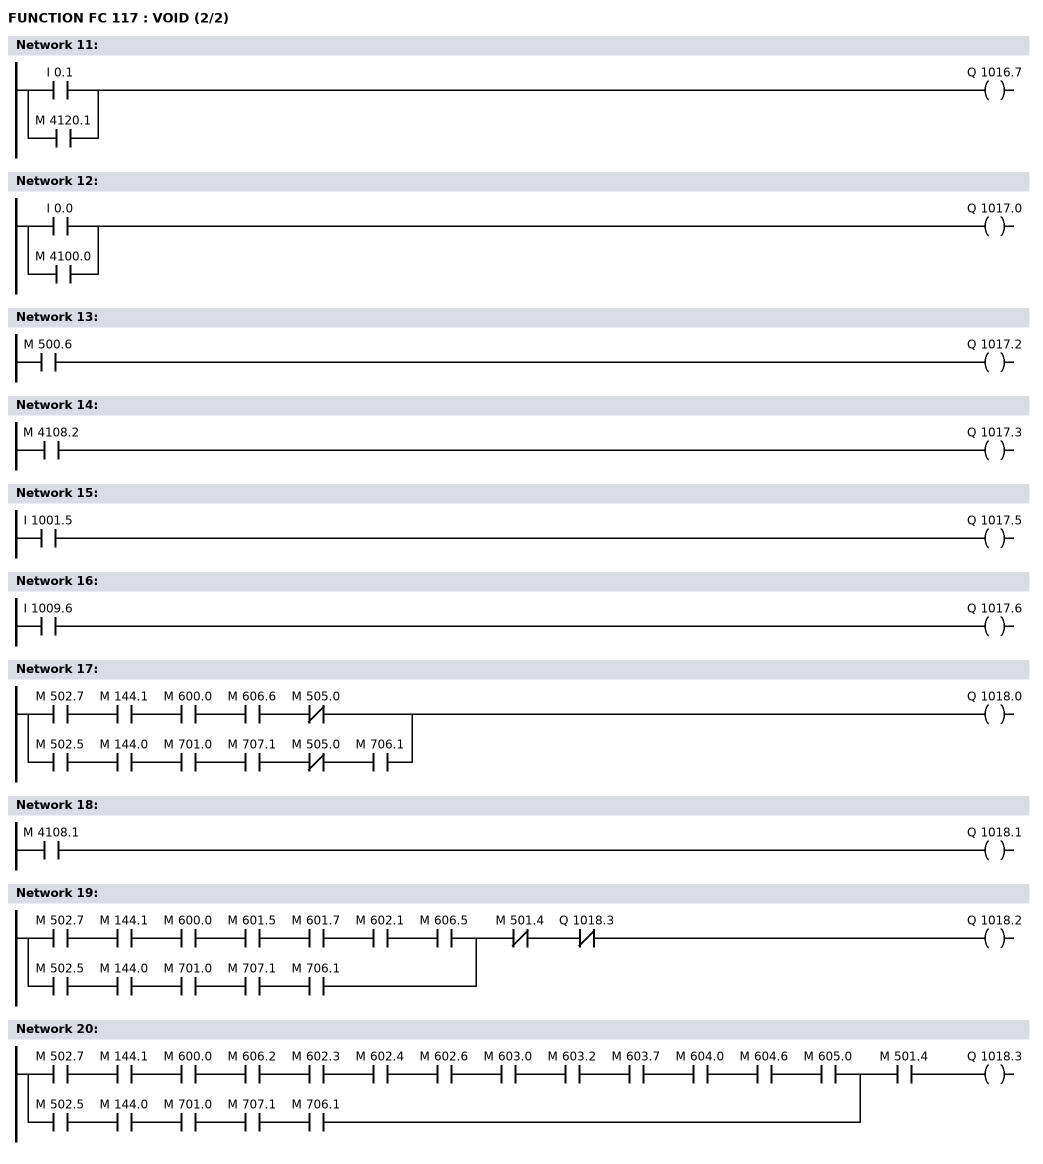

      O     I      0.1;
      O     M   4120.1;
      =     Q   1016.7;
NETWORK
TITLE =

      O     I      0.0;
      O     M   4100.0;
      =     Q   1017.0;
NETWORK
TITLE =

      A     M    500.6;
      =     Q   1017.2;
NETWORK
TITLE =

      A     M   4108.2;
      =     Q   1017.3;
NETWORK
TITLE =

      A     I   1001.5;
      =     Q   1017.5;
NETWORK
TITLE =

      A     I   1009.6;
      =     Q   1017.6;
NETWORK
TITLE =

      A     M    502.7;
      A     M    144.1;
      A     M    600.0;
      A     M    606.6;
      AN    M    505.0;
      O     ;
      A     M    502.5;
      A     M    144.0;
      A     M    701.0;
      A     M    707.1;
      AN    M    505.0;
      A     M    706.1;
      =     Q   1018.0;
NETWORK
TITLE =

      A     M   4108.1;
      =     Q   1018.1;
NETWORK
TITLE =

      A(    ;
      A     M    502.7;
      A     M    144.1;
      A     M    600.0;
      A     M    601.5;
      A     M    601.7;
      A     M    602.1;
      A     M    606.5;
      O     ;
      A     M    502.5;
      A     M    144.0;
      A     M    701.0;
      A     M    707.1;
      A     M    706.1;
      )     ;
      AN    M    501.4;
      AN    Q   1018.3;
      =     Q   1018.2;
NETWORK
TITLE =

      A(    ;
      A     M    502.7;
      A     M    144.1;
      A     M    600.0;
      A     M    606.2;
      A     M    602.3;
      A     M    602.4;
      A     M    602.6;
      A     M    603.0;
      A     M    603.2;
      A     M    603.7;
      A     M    604.0;
      A     M    604.6;
      A     M    605.0;
      O     ;
      A     M    502.5;
      A     M    144.0;
      A     M    701.0;
      A     M    707.1;
      A     M    706.1;
      )     ;
      A     M    501.4;
      =     Q   1018.3;
END_FUNCTION

FUNCTION_BLOCK FB 120
TITLE =
VERSION : 0.1


VAR
  S706_MODE : FB 402;
END_VAR
BEGIN
NETWORK
TITLE =
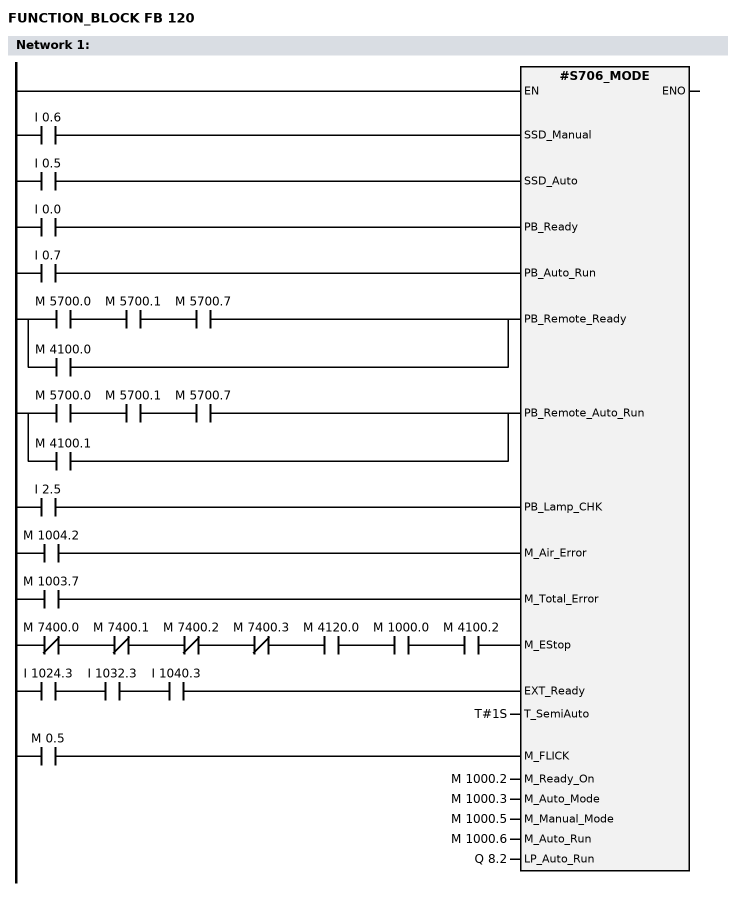

      A     I      0.6;
      =     L      0.0;
      BLD   103;
      A     I      0.5;
      =     L      0.1;
      BLD   103;
      A     I      0.0;
      =     L      0.2;
      BLD   103;
      A     I      0.7;
      =     L      0.3;
      BLD   103;
      A(    ;
      A     M   5700.0;
      A     M   5700.1;
      A     M   5700.7;
      O     M   4100.0;
      )     ;
      =     L      0.4;
      BLD   103;
      A(    ;
      A     M   5700.0;
      A     M   5700.1;
      A     M   5700.7;
      O     M   4100.1;
      )     ;
      =     L      0.5;
      BLD   103;
      A     I      2.5;
      =     L      0.6;
      BLD   103;
      A     M   1004.2;
      =     L      0.7;
      BLD   103;
      A     M   1003.7;
      =     L      1.1;
      BLD   103;
      AN    M   7400.0;
      AN    M   7400.1;
      AN    M   7400.2;
      AN    M   7400.3;
      A     M   4120.0;
      A     M   1000.0;
      A     M   4100.2;
      =     L      1.2;
      BLD   103;
      A     I   1024.3;
      A     I   1032.3;
      A     I   1040.3;
      =     L      1.3;
      BLD   103;
      A     M      0.5;
      =     L      1.5;
      BLD   103;
      CALL #S706_MODE (
           SSD_Manual               := L      0.0,
           SSD_Auto                 := L      0.1,
           PB_Ready                 := L      0.2,
           PB_Auto_Run              := L      0.3,
           PB_Remote_Ready          := L      0.4,
           PB_Remote_Auto_Run       := L      0.5,
           PB_Lamp_CHK              := L      0.6,
           M_Air_Error              := L      0.7,
           M_Total_Error            := L      1.1,
           M_EStop                  := L      1.2,
           EXT_Ready                := L      1.3,
           T_SemiAuto               := T#1S,
           M_FLICK                  := L      1.5,
           M_Ready_On               := M   1000.2,
           M_Auto_Mode              := M   1000.3,
           M_Manual_Mode            := M   1000.5,
           M_Auto_Run               := M   1000.6,
           LP_Auto_Run              := Q      8.2);
      NOP   0;
END_FUNCTION_BLOCK

DATA_BLOCK DB 120
TITLE =
VERSION : 0.0

 FB 120
BEGIN
   S706_MODE.SSD_Manual := FALSE;
   S706_MODE.SSD_Auto := TRUE;
   S706_MODE.PB_Ready := FALSE;
   S706_MODE.PB_Auto_Run := FALSE;
   S706_MODE.PB_Remote_Ready := FALSE;
   S706_MODE.PB_Remote_Auto_Run := FALSE;
   S706_MODE.PB_Lamp_CHK := FALSE;
   S706_MODE.M_Air_Error := FALSE;
   S706_MODE.M_Water_Error := FALSE;
   S706_MODE.M_Total_Error := FALSE;
   S706_MODE.M_EStop := TRUE;
   S706_MODE.EXT_Ready := TRUE;
   S706_MODE.EXT_Auto := FALSE;
   S706_MODE.T_SemiAuto := T#1S;
   S706_MODE.M_FLICK := TRUE;
   S706_MODE.M_Ready_On := TRUE;
   S706_MODE.M_Auto_Mode := TRUE;
   S706_MODE.M_SemiAuto_Mode := FALSE;
   S706_MODE.M_Manual_Mode := FALSE;
   S706_MODE.M_Auto_Run := TRUE;
   S706_MODE.LP_Ready_On := TRUE;
   S706_MODE.LP_Auto_Run := TRUE;
   S706_MODE.AUTO_MODE_DELAY.IN := FALSE;
   S706_MODE.AUTO_MODE_DELAY.PT := T#0MS;
   S706_MODE.AUTO_MODE_DELAY.Q := FALSE;
   S706_MODE.AUTO_MODE_DELAY.ET := T#0MS;
   S706_MODE.AUTO_MODE_DELAY.STATE := B#16#0;
   S706_MODE.AUTO_MODE_DELAY.STIME := T#0MS;
   S706_MODE.AUTO_MODE_DELAY.ATIME := T#0MS;
   S706_MODE.SEMI_AUTO_DELAY.IN := FALSE;
   S706_MODE.SEMI_AUTO_DELAY.PT := T#1S;
   S706_MODE.SEMI_AUTO_DELAY.Q := FALSE;
   S706_MODE.SEMI_AUTO_DELAY.ET := T#0MS;
   S706_MODE.SEMI_AUTO_DELAY.STATE := B#16#0;
   S706_MODE.SEMI_AUTO_DELAY.STIME := T#3D5H44M23S926MS;
   S706_MODE.SEMI_AUTO_DELAY.ATIME := T#3D5H44M23S950MS;
   S706_MODE.MANUAL_DELAY.IN := FALSE;
   S706_MODE.MANUAL_DELAY.PT := T#0MS;
   S706_MODE.MANUAL_DELAY.Q := FALSE;
   S706_MODE.MANUAL_DELAY.ET := T#0MS;
   S706_MODE.MANUAL_DELAY.STATE := B#16#0;
   S706_MODE.MANUAL_DELAY.STIME := T#0MS;
   S706_MODE.MANUAL_DELAY.ATIME := T#0MS;
END_DATA_BLOCK

FUNCTION FC 120 : VOID
TITLE =
VERSION : 0.1

BEGIN
NETWORK
TITLE =
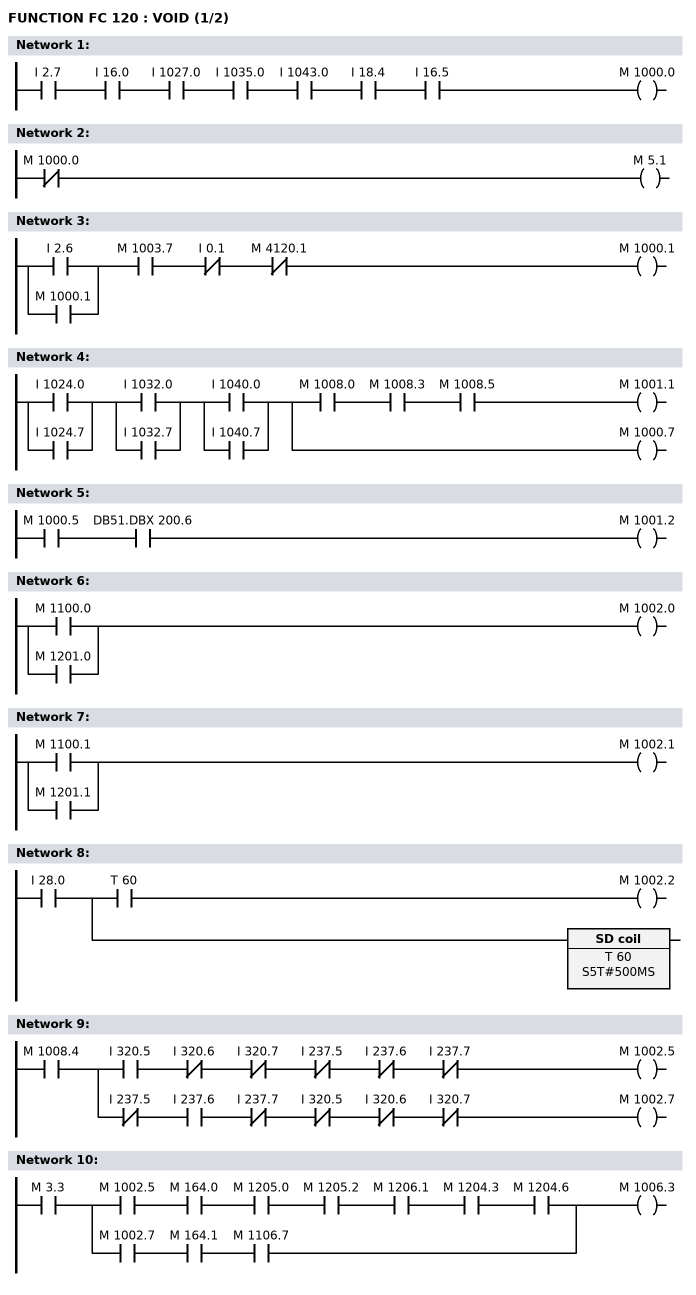

      A     I      2.7;
      A     I     16.0;
      A     I   1027.0;
      A     I   1035.0;
      A     I   1043.0;
      A     I     18.4;
      A     I     16.5;
      =     M   1000.0;
NETWORK
TITLE =

      AN    M   1000.0;
      =     M      5.1;
NETWORK
TITLE =

      A(    ;
      O     I      2.6;
      O     M   1000.1;
      )     ;
      A     M   1003.7;
      AN    I      0.1;
      AN    M   4120.1;
      =     M   1000.1;
NETWORK
TITLE =

      A(    ;
      O     I   1024.0;
      O     I   1024.7;
      )     ;
      A(    ;
      O     I   1032.0;
      O     I   1032.7;
      )     ;
      A(    ;
      O     I   1040.0;
      O     I   1040.7;
      )     ;
      =     L      0.0;
      A     L      0.0;
      A     M   1008.0;
      A     M   1008.3;
      A     M   1008.5;
      =     M   1001.1;
      A     L      0.0;
      BLD   102;
      =     M   1000.7;
NETWORK
TITLE =

      A     M   1000.5;
      A     DB51.DBX  200.6;
      =     M   1001.2;
NETWORK
TITLE =

      O     M   1100.0;
      O     M   1201.0;
      =     M   1002.0;
NETWORK
TITLE =

      O     M   1100.1;
      O     M   1201.1;
      =     M   1002.1;
NETWORK
TITLE =

      A     I     28.0;
      =     L      0.0;
      A     L      0.0;
      A     T     60;
      =     M   1002.2;
      A     L      0.0;
      BLD   102;
      L     S5T#500MS;
      SD    T     60;
NETWORK
TITLE =

      A     M   1008.4;
      =     L      0.0;
      A     L      0.0;
      A     I    320.5;
      AN    I    320.6;
      AN    I    320.7;
      AN    I    237.5;
      AN    I    237.6;
      AN    I    237.7;
      =     M   1002.5;
      A     L      0.0;
      AN    I    237.5;
      A     I    237.6;
      AN    I    237.7;
      AN    I    320.5;
      AN    I    320.6;
      AN    I    320.7;
      =     M   1002.7;
NETWORK
TITLE =

      A     M      3.3;
      A(    ;
      A     M   1002.5;
      A     M    164.0;
      A     M   1205.0;
      A     M   1205.2;
      A     M   1206.1;
      A     M   1204.3;
      A     M   1204.6;
      O     ;
      A     M   1002.7;
      A     M    164.1;
      A     M   1106.7;
      )     ;
      =     M   1006.3;
NETWORK
TITLE =
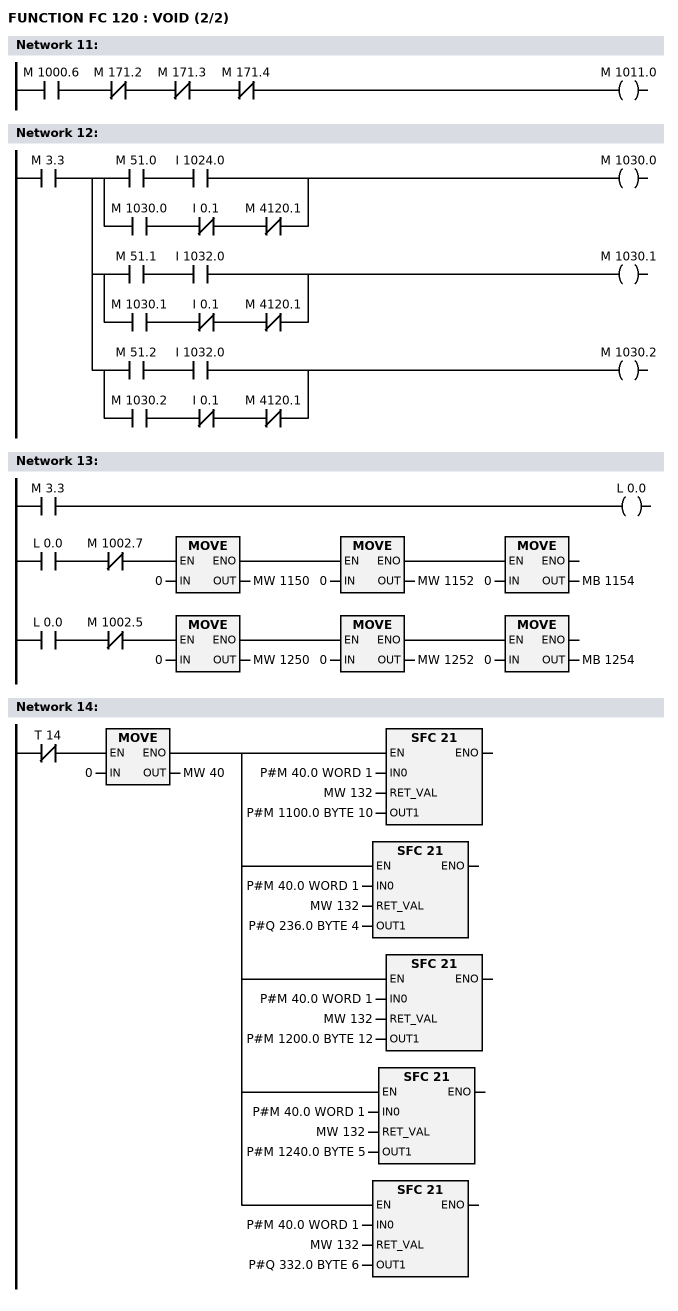

      A     M   1000.6;
      AN    M    171.2;
      AN    M    171.3;
      AN    M    171.4;
      =     M   1011.0;
NETWORK
TITLE =

      A     M      3.3;
      =     L      0.0;
      A     L      0.0;
      A(    ;
      A     M     51.0;
      A     I   1024.0;
      O     ;
      A     M   1030.0;
      AN    I      0.1;
      AN    M   4120.1;
      )     ;
      =     M   1030.0;
      A     L      0.0;
      A(    ;
      A     M     51.1;
      A     I   1032.0;
      O     ;
      A     M   1030.1;
      AN    I      0.1;
      AN    M   4120.1;
      )     ;
      =     M   1030.1;
      A     L      0.0;
      A(    ;
      A     M     51.2;
      A     I   1032.0;
      O     ;
      A     M   1030.2;
      AN    I      0.1;
      AN    M   4120.1;
      )     ;
      =     M   1030.2;
NETWORK
TITLE =

      A     M      3.3;
      =     L      0.0;
      A(    ;
      A(    ;
      A     L      0.0;
      AN    M   1002.7;
      JNB   _001;
      L     0;
      T     MW  1150;
      SET   ;
      SAVE  ;
      CLR   ;
_001: A     BR;
      )     ;
      JNB   _002;
      L     0;
      T     MW  1152;
      SET   ;
      SAVE  ;
      CLR   ;
_002: A     BR;
      )     ;
      JNB   _003;
      L     0;
      T     MB  1154;
_003: NOP   0;
      A(    ;
      A(    ;
      A     L      0.0;
      AN    M   1002.5;
      JNB   _004;
      L     0;
      T     MW  1250;
      SET   ;
      SAVE  ;
      CLR   ;
_004: A     BR;
      )     ;
      JNB   _005;
      L     0;
      T     MW  1252;
      SET   ;
      SAVE  ;
      CLR   ;
_005: A     BR;
      )     ;
      JNB   _006;
      L     0;
      T     MB  1254;
_006: NOP   0;
NETWORK
TITLE =

      AN    T     14;
      JNB   _007;
      L     0;
      T     MW    40;
      SET   ;
      SAVE  ;
      CLR   ;
_007: A     BR;
      =     L      0.0;
      A     L      0.0;
      JNB   _008;
      CALL SFC   21 (
           IN0                      := P#M 40.0 WORD 1,
           RET_VAL                  := MW   132,
           OUT1                     := P#M 1100.0 BYTE 10);
_008: NOP   0;
      A     L      0.0;
      JNB   _009;
      CALL SFC   21 (
           IN0                      := P#M 40.0 WORD 1,
           RET_VAL                  := MW   132,
           OUT1                     := P#Q 236.0 BYTE 4);
_009: NOP   0;
      A     L      0.0;
      JNB   _00a;
      CALL SFC   21 (
           IN0                      := P#M 40.0 WORD 1,
           RET_VAL                  := MW   132,
           OUT1                     := P#M 1200.0 BYTE 12);
_00a: NOP   0;
      A     L      0.0;
      JNB   _00b;
      CALL SFC   21 (
           IN0                      := P#M 40.0 WORD 1,
           RET_VAL                  := MW   132,
           OUT1                     := P#M 1240.0 BYTE 5);
_00b: NOP   0;
      A     L      0.0;
      JNB   _00c;
      CALL SFC   21 (
           IN0                      := P#M 40.0 WORD 1,
           RET_VAL                  := MW   132,
           OUT1                     := P#Q 332.0 BYTE 6);
_00c: NOP   0;
END_FUNCTION

FUNCTION_BLOCK FB 121
TITLE =
VERSION : 0.1


VAR
  S706_HOOK_PIN : FB 424;
  S706_DC_LOCK : FB 424;
  S706_ELE : FB 424;
  S706_AIR_ELE : FB 424;
END_VAR
BEGIN
NETWORK
TITLE =
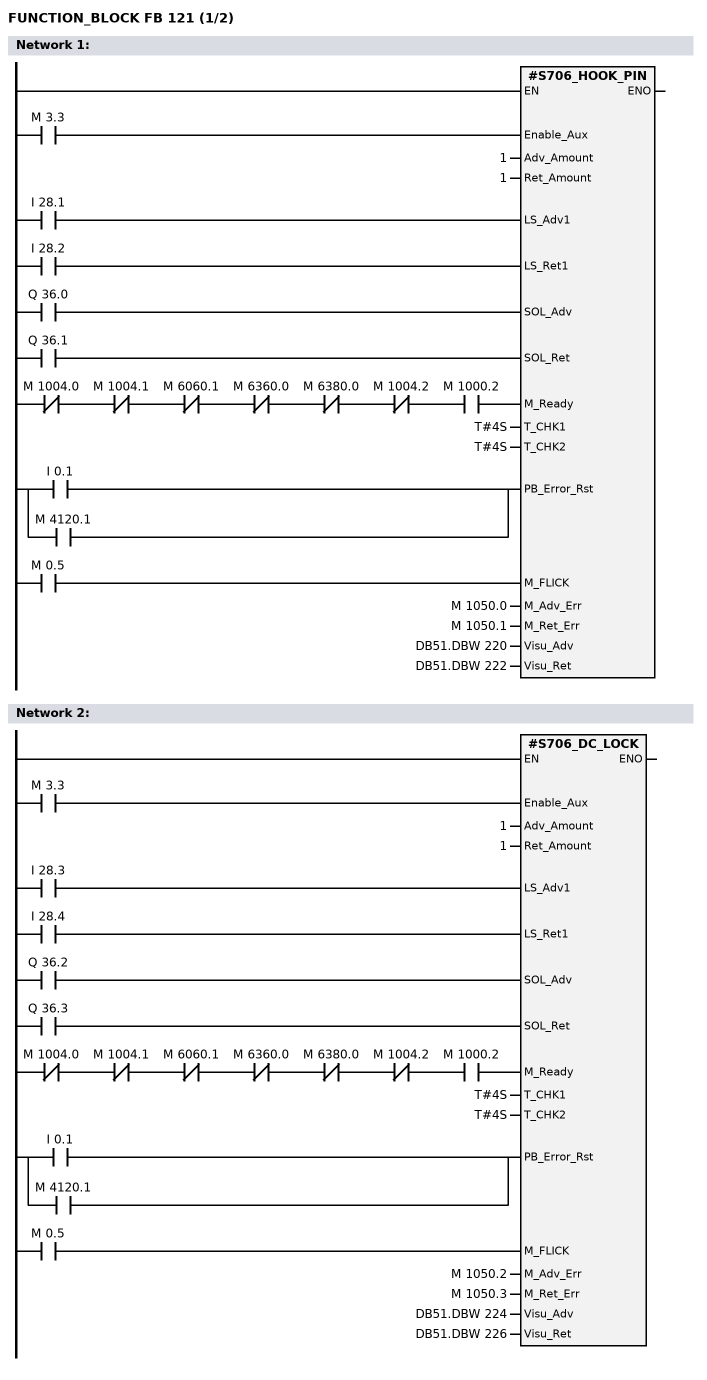

      A     M      3.3;
      =     L      0.0;
      BLD   103;
      A     I     28.1;
      =     L      0.1;
      BLD   103;
      A     I     28.2;
      =     L      0.2;
      BLD   103;
      A     Q     36.0;
      =     L      1.1;
      BLD   103;
      A     Q     36.1;
      =     L      1.2;
      BLD   103;
      AN    M   1004.0;
      AN    M   1004.1;
      AN    M   6060.1;
      AN    M   6360.0;
      AN    M   6380.0;
      AN    M   1004.2;
      A     M   1000.2;
      =     L      1.3;
      BLD   103;
      A(    ;
      O     I      0.1;
      O     M   4120.1;
      )     ;
      =     L      1.5;
      BLD   103;
      A     M      0.5;
      =     L      1.6;
      BLD   103;
      CALL #S706_HOOK_PIN (
           Enable_Aux               := L      0.0,
           Adv_Amount               := 1,
           Ret_Amount               := 1,
           LS_Adv1                  := L      0.1,
           LS_Ret1                  := L      0.2,
           SOL_Adv                  := L      1.1,
           SOL_Ret                  := L      1.2,
           M_Ready                  := L      1.3,
           T_CHK1                   := T#4S,
           T_CHK2                   := T#4S,
           PB_Error_Rst             := L      1.5,
           M_FLICK                  := L      1.6,
           M_Adv_Err                := M   1050.0,
           M_Ret_Err                := M   1050.1,
           Visu_Adv                 := DB51.DBW  220,
           Visu_Ret                 := DB51.DBW  222);
      NOP   0;
NETWORK
TITLE =

      A     M      3.3;
      =     L      0.0;
      BLD   103;
      A     I     28.3;
      =     L      0.1;
      BLD   103;
      A     I     28.4;
      =     L      0.2;
      BLD   103;
      A     Q     36.2;
      =     L      1.1;
      BLD   103;
      A     Q     36.3;
      =     L      1.2;
      BLD   103;
      AN    M   1004.0;
      AN    M   1004.1;
      AN    M   6060.1;
      AN    M   6360.0;
      AN    M   6380.0;
      AN    M   1004.2;
      A     M   1000.2;
      =     L      1.3;
      BLD   103;
      A(    ;
      O     I      0.1;
      O     M   4120.1;
      )     ;
      =     L      1.5;
      BLD   103;
      A     M      0.5;
      =     L      1.6;
      BLD   103;
      CALL #S706_DC_LOCK (
           Enable_Aux               := L      0.0,
           Adv_Amount               := 1,
           Ret_Amount               := 1,
           LS_Adv1                  := L      0.1,
           LS_Ret1                  := L      0.2,
           SOL_Adv                  := L      1.1,
           SOL_Ret                  := L      1.2,
           M_Ready                  := L      1.3,
           T_CHK1                   := T#4S,
           T_CHK2                   := T#4S,
           PB_Error_Rst             := L      1.5,
           M_FLICK                  := L      1.6,
           M_Adv_Err                := M   1050.2,
           M_Ret_Err                := M   1050.3,
           Visu_Adv                 := DB51.DBW  224,
           Visu_Ret                 := DB51.DBW  226);
      NOP   0;
NETWORK
TITLE =
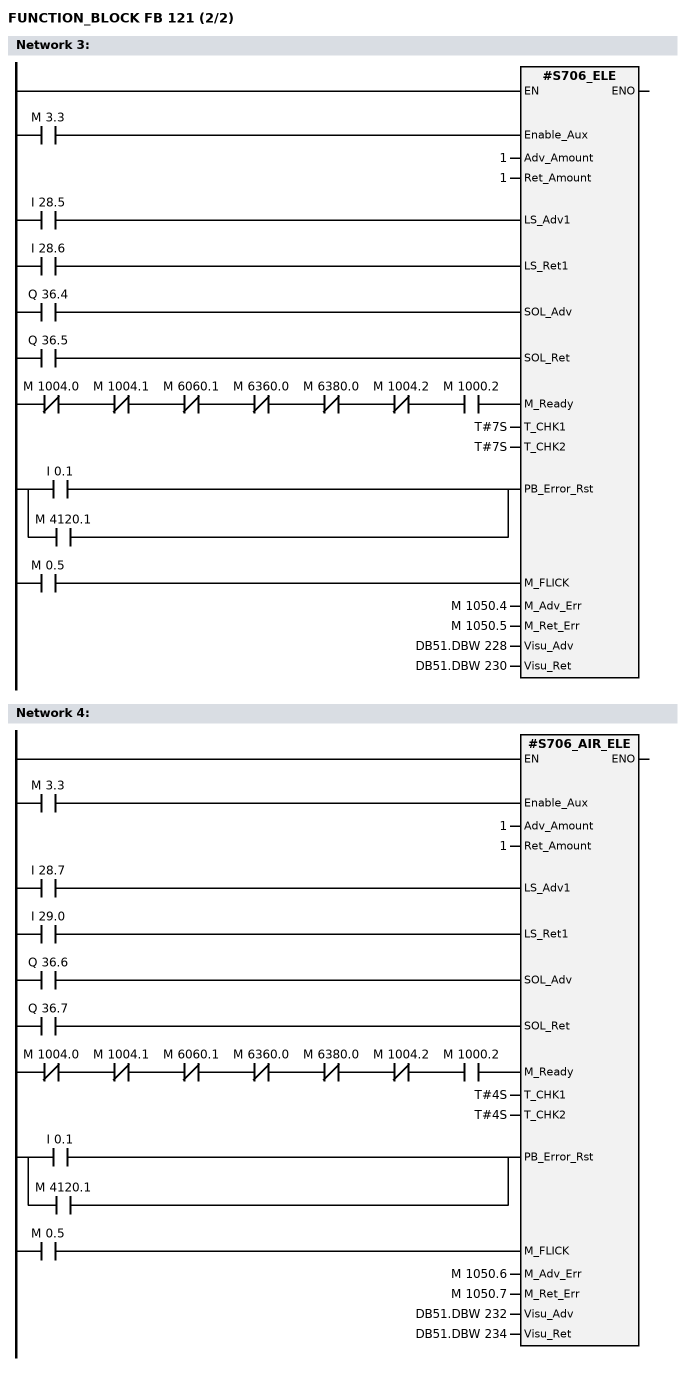

      A     M      3.3;
      =     L      0.0;
      BLD   103;
      A     I     28.5;
      =     L      0.1;
      BLD   103;
      A     I     28.6;
      =     L      0.2;
      BLD   103;
      A     Q     36.4;
      =     L      1.1;
      BLD   103;
      A     Q     36.5;
      =     L      1.2;
      BLD   103;
      AN    M   1004.0;
      AN    M   1004.1;
      AN    M   6060.1;
      AN    M   6360.0;
      AN    M   6380.0;
      AN    M   1004.2;
      A     M   1000.2;
      =     L      1.3;
      BLD   103;
      A(    ;
      O     I      0.1;
      O     M   4120.1;
      )     ;
      =     L      1.5;
      BLD   103;
      A     M      0.5;
      =     L      1.6;
      BLD   103;
      CALL #S706_ELE (
           Enable_Aux               := L      0.0,
           Adv_Amount               := 1,
           Ret_Amount               := 1,
           LS_Adv1                  := L      0.1,
           LS_Ret1                  := L      0.2,
           SOL_Adv                  := L      1.1,
           SOL_Ret                  := L      1.2,
           M_Ready                  := L      1.3,
           T_CHK1                   := T#7S,
           T_CHK2                   := T#7S,
           PB_Error_Rst             := L      1.5,
           M_FLICK                  := L      1.6,
           M_Adv_Err                := M   1050.4,
           M_Ret_Err                := M   1050.5,
           Visu_Adv                 := DB51.DBW  228,
           Visu_Ret                 := DB51.DBW  230);
      NOP   0;
NETWORK
TITLE =

      A     M      3.3;
      =     L      0.0;
      BLD   103;
      A     I     28.7;
      =     L      0.1;
      BLD   103;
      A     I     29.0;
      =     L      0.2;
      BLD   103;
      A     Q     36.6;
      =     L      1.1;
      BLD   103;
      A     Q     36.7;
      =     L      1.2;
      BLD   103;
      AN    M   1004.0;
      AN    M   1004.1;
      AN    M   6060.1;
      AN    M   6360.0;
      AN    M   6380.0;
      AN    M   1004.2;
      A     M   1000.2;
      =     L      1.3;
      BLD   103;
      A(    ;
      O     I      0.1;
      O     M   4120.1;
      )     ;
      =     L      1.5;
      BLD   103;
      A     M      0.5;
      =     L      1.6;
      BLD   103;
      CALL #S706_AIR_ELE (
           Enable_Aux               := L      0.0,
           Adv_Amount               := 1,
           Ret_Amount               := 1,
           LS_Adv1                  := L      0.1,
           LS_Ret1                  := L      0.2,
           SOL_Adv                  := L      1.1,
           SOL_Ret                  := L      1.2,
           M_Ready                  := L      1.3,
           T_CHK1                   := T#4S,
           T_CHK2                   := T#4S,
           PB_Error_Rst             := L      1.5,
           M_FLICK                  := L      1.6,
           M_Adv_Err                := M   1050.6,
           M_Ret_Err                := M   1050.7,
           Visu_Adv                 := DB51.DBW  232,
           Visu_Ret                 := DB51.DBW  234);
      NOP   0;
END_FUNCTION_BLOCK

DATA_BLOCK DB 121
TITLE =
VERSION : 0.0

 FB 121
BEGIN
   S706_HOOK_PIN.Enable_Aux := TRUE;
   S706_HOOK_PIN.Adv_Amount := 1;
   S706_HOOK_PIN.Ret_Amount := 1;
   S706_HOOK_PIN.LS_Adv1 := FALSE;
   S706_HOOK_PIN.LS_Ret1 := TRUE;
   S706_HOOK_PIN.LS_Adv2 := FALSE;
   S706_HOOK_PIN.LS_Ret2 := FALSE;
   S706_HOOK_PIN.LS_Adv3 := FALSE;
   S706_HOOK_PIN.LS_Ret3 := FALSE;
   S706_HOOK_PIN.LS_Adv4 := FALSE;
   S706_HOOK_PIN.LS_Ret4 := FALSE;
   S706_HOOK_PIN.SOL_Adv := FALSE;
   S706_HOOK_PIN.SOL_Ret := FALSE;
   S706_HOOK_PIN.M_Ready := TRUE;
   S706_HOOK_PIN.T_CHK1 := T#4S;
   S706_HOOK_PIN.T_CHK2 := T#4S;
   S706_HOOK_PIN.PB_Lamp_CHK := FALSE;
   S706_HOOK_PIN.PB_Error_Rst := FALSE;
   S706_HOOK_PIN.M_FLICK := TRUE;
   S706_HOOK_PIN.M_Adv_Err := FALSE;
   S706_HOOK_PIN.M_Ret_Err := FALSE;
   S706_HOOK_PIN.LP_Adv := FALSE;
   S706_HOOK_PIN.LP_Ret := TRUE;
   S706_HOOK_PIN.Visu_Adv := W#16#0;
   S706_HOOK_PIN.Visu_Ret := W#16#300;
   S706_HOOK_PIN.Error_T1.IN := FALSE;
   S706_HOOK_PIN.Error_T1.PT := T#4S;
   S706_HOOK_PIN.Error_T1.Q := FALSE;
   S706_HOOK_PIN.Error_T1.ET := T#0MS;
   S706_HOOK_PIN.Error_T1.STATE := B#16#0;
   S706_HOOK_PIN.Error_T1.STIME := T#23D5H8M43S363MS;
   S706_HOOK_PIN.Error_T1.ATIME := T#23D5H8M43S776MS;
   S706_HOOK_PIN.Error_T2.IN := FALSE;
   S706_HOOK_PIN.Error_T2.PT := T#4S;
   S706_HOOK_PIN.Error_T2.Q := FALSE;
   S706_HOOK_PIN.Error_T2.ET := T#0MS;
   S706_HOOK_PIN.Error_T2.STATE := B#16#0;
   S706_HOOK_PIN.Error_T2.STIME := T#0MS;
   S706_HOOK_PIN.Error_T2.ATIME := T#0MS;
   S706_HOOK_PIN.CHK_Aux1 := FALSE;
   S706_HOOK_PIN.CHK_Aux2 := FALSE;
   S706_HOOK_PIN.Error_T1_DN := FALSE;
   S706_HOOK_PIN.Error_T2_DN := FALSE;
   S706_HOOK_PIN.Adv_Memo := FALSE;
   S706_HOOK_PIN.Visu_Adv_Arr[0] := FALSE;
   S706_HOOK_PIN.Visu_Adv_Arr[1] := FALSE;
   S706_HOOK_PIN.Visu_Adv_Arr[2] := FALSE;
   S706_HOOK_PIN.Visu_Adv_Arr[3] := FALSE;
   S706_HOOK_PIN.Visu_Adv_Arr[4] := FALSE;
   S706_HOOK_PIN.Visu_Adv_Arr[5] := FALSE;
   S706_HOOK_PIN.Visu_Adv_Arr[6] := FALSE;
   S706_HOOK_PIN.Visu_Adv_Arr[7] := FALSE;
   S706_HOOK_PIN.Visu_Adv_Arr[8] := FALSE;
   S706_HOOK_PIN.Visu_Adv_Arr[9] := FALSE;
   S706_HOOK_PIN.Visu_Adv_Arr[10] := FALSE;
   S706_HOOK_PIN.Visu_Adv_Arr[11] := FALSE;
   S706_HOOK_PIN.Visu_Adv_Arr[12] := FALSE;
   S706_HOOK_PIN.Visu_Adv_Arr[13] := FALSE;
   S706_HOOK_PIN.Visu_Adv_Arr[14] := FALSE;
   S706_HOOK_PIN.Visu_Adv_Arr[15] := FALSE;
   S706_HOOK_PIN.Visu_Ret_Arr[0] := TRUE;
   S706_HOOK_PIN.Visu_Ret_Arr[1] := TRUE;
   S706_HOOK_PIN.Visu_Ret_Arr[2] := FALSE;
   S706_HOOK_PIN.Visu_Ret_Arr[3] := FALSE;
   S706_HOOK_PIN.Visu_Ret_Arr[4] := FALSE;
   S706_HOOK_PIN.Visu_Ret_Arr[5] := FALSE;
   S706_HOOK_PIN.Visu_Ret_Arr[6] := FALSE;
   S706_HOOK_PIN.Visu_Ret_Arr[7] := FALSE;
   S706_HOOK_PIN.Visu_Ret_Arr[8] := FALSE;
   S706_HOOK_PIN.Visu_Ret_Arr[9] := FALSE;
   S706_HOOK_PIN.Visu_Ret_Arr[10] := FALSE;
   S706_HOOK_PIN.Visu_Ret_Arr[11] := FALSE;
   S706_HOOK_PIN.Visu_Ret_Arr[12] := FALSE;
   S706_HOOK_PIN.Visu_Ret_Arr[13] := FALSE;
   S706_HOOK_PIN.Visu_Ret_Arr[14] := FALSE;
   S706_HOOK_PIN.Visu_Ret_Arr[15] := FALSE;
   S706_HOOK_PIN.BLK_Move_Ret := 0;
   S706_HOOK_PIN.Enable := TRUE;
   S706_HOOK_PIN.Adv_End := FALSE;
   S706_HOOK_PIN.Ret_End := TRUE;
   S706_DC_LOCK.Enable_Aux := TRUE;
   S706_DC_LOCK.Adv_Amount := 1;
   S706_DC_LOCK.Ret_Amount := 1;
   S706_DC_LOCK.LS_Adv1 := TRUE;
   S706_DC_LOCK.LS_Ret1 := FALSE;
   S706_DC_LOCK.LS_Adv2 := FALSE;
   S706_DC_LOCK.LS_Ret2 := FALSE;
   S706_DC_LOCK.LS_Adv3 := FALSE;
   S706_DC_LOCK.LS_Ret3 := FALSE;
   S706_DC_LOCK.LS_Adv4 := FALSE;
   S706_DC_LOCK.LS_Ret4 := FALSE;
   S706_DC_LOCK.SOL_Adv := FALSE;
   S706_DC_LOCK.SOL_Ret := FALSE;
   S706_DC_LOCK.M_Ready := TRUE;
   S706_DC_LOCK.T_CHK1 := T#4S;
   S706_DC_LOCK.T_CHK2 := T#4S;
   S706_DC_LOCK.PB_Lamp_CHK := FALSE;
   S706_DC_LOCK.PB_Error_Rst := FALSE;
   S706_DC_LOCK.M_FLICK := TRUE;
   S706_DC_LOCK.M_Adv_Err := FALSE;
   S706_DC_LOCK.M_Ret_Err := FALSE;
   S706_DC_LOCK.LP_Adv := TRUE;
   S706_DC_LOCK.LP_Ret := FALSE;
   S706_DC_LOCK.Visu_Adv := W#16#300;
   S706_DC_LOCK.Visu_Ret := W#16#0;
   S706_DC_LOCK.Error_T1.IN := FALSE;
   S706_DC_LOCK.Error_T1.PT := T#4S;
   S706_DC_LOCK.Error_T1.Q := FALSE;
   S706_DC_LOCK.Error_T1.ET := T#0MS;
   S706_DC_LOCK.Error_T1.STATE := B#16#0;
   S706_DC_LOCK.Error_T1.STIME := T#23D5H8M43S363MS;
   S706_DC_LOCK.Error_T1.ATIME := T#23D5H8M43S848MS;
   S706_DC_LOCK.Error_T2.IN := FALSE;
   S706_DC_LOCK.Error_T2.PT := T#4S;
   S706_DC_LOCK.Error_T2.Q := FALSE;
   S706_DC_LOCK.Error_T2.ET := T#0MS;
   S706_DC_LOCK.Error_T2.STATE := B#16#0;
   S706_DC_LOCK.Error_T2.STIME := T#0MS;
   S706_DC_LOCK.Error_T2.ATIME := T#0MS;
   S706_DC_LOCK.CHK_Aux1 := FALSE;
   S706_DC_LOCK.CHK_Aux2 := FALSE;
   S706_DC_LOCK.Error_T1_DN := FALSE;
   S706_DC_LOCK.Error_T2_DN := FALSE;
   S706_DC_LOCK.Adv_Memo := TRUE;
   S706_DC_LOCK.Visu_Adv_Arr[0] := TRUE;
   S706_DC_LOCK.Visu_Adv_Arr[1] := TRUE;
   S706_DC_LOCK.Visu_Adv_Arr[2] := FALSE;
   S706_DC_LOCK.Visu_Adv_Arr[3] := FALSE;
   S706_DC_LOCK.Visu_Adv_Arr[4] := FALSE;
   S706_DC_LOCK.Visu_Adv_Arr[5] := FALSE;
   S706_DC_LOCK.Visu_Adv_Arr[6] := FALSE;
   S706_DC_LOCK.Visu_Adv_Arr[7] := FALSE;
   S706_DC_LOCK.Visu_Adv_Arr[8] := FALSE;
   S706_DC_LOCK.Visu_Adv_Arr[9] := FALSE;
   S706_DC_LOCK.Visu_Adv_Arr[10] := FALSE;
   S706_DC_LOCK.Visu_Adv_Arr[11] := FALSE;
   S706_DC_LOCK.Visu_Adv_Arr[12] := FALSE;
   S706_DC_LOCK.Visu_Adv_Arr[13] := FALSE;
   S706_DC_LOCK.Visu_Adv_Arr[14] := FALSE;
   S706_DC_LOCK.Visu_Adv_Arr[15] := FALSE;
   S706_DC_LOCK.Visu_Ret_Arr[0] := FALSE;
   S706_DC_LOCK.Visu_Ret_Arr[1] := FALSE;
   S706_DC_LOCK.Visu_Ret_Arr[2] := FALSE;
   S706_DC_LOCK.Visu_Ret_Arr[3] := FALSE;
   S706_DC_LOCK.Visu_Ret_Arr[4] := FALSE;
   S706_DC_LOCK.Visu_Ret_Arr[5] := FALSE;
   S706_DC_LOCK.Visu_Ret_Arr[6] := FALSE;
   S706_DC_LOCK.Visu_Ret_Arr[7] := FALSE;
   S706_DC_LOCK.Visu_Ret_Arr[8] := FALSE;
   S706_DC_LOCK.Visu_Ret_Arr[9] := FALSE;
   S706_DC_LOCK.Visu_Ret_Arr[10] := FALSE;
   S706_DC_LOCK.Visu_Ret_Arr[11] := FALSE;
   S706_DC_LOCK.Visu_Ret_Arr[12] := FALSE;
   S706_DC_LOCK.Visu_Ret_Arr[13] := FALSE;
   S706_DC_LOCK.Visu_Ret_Arr[14] := FALSE;
   S706_DC_LOCK.Visu_Ret_Arr[15] := FALSE;
   S706_DC_LOCK.BLK_Move_Ret := 0;
   S706_DC_LOCK.Enable := TRUE;
   S706_DC_LOCK.Adv_End := TRUE;
   S706_DC_LOCK.Ret_End := FALSE;
   S706_ELE.Enable_Aux := TRUE;
   S706_ELE.Adv_Amount := 1;
   S706_ELE.Ret_Amount := 1;
   S706_ELE.LS_Adv1 := TRUE;
   S706_ELE.LS_Ret1 := FALSE;
   S706_ELE.LS_Adv2 := FALSE;
   S706_ELE.LS_Ret2 := FALSE;
   S706_ELE.LS_Adv3 := FALSE;
   S706_ELE.LS_Ret3 := FALSE;
   S706_ELE.LS_Adv4 := FALSE;
   S706_ELE.LS_Ret4 := FALSE;
   S706_ELE.SOL_Adv := FALSE;
   S706_ELE.SOL_Ret := FALSE;
   S706_ELE.M_Ready := TRUE;
   S706_ELE.T_CHK1 := T#7S;
   S706_ELE.T_CHK2 := T#7S;
   S706_ELE.PB_Lamp_CHK := FALSE;
   S706_ELE.PB_Error_Rst := FALSE;
   S706_ELE.M_FLICK := TRUE;
   S706_ELE.M_Adv_Err := FALSE;
   S706_ELE.M_Ret_Err := FALSE;
   S706_ELE.LP_Adv := TRUE;
   S706_ELE.LP_Ret := FALSE;
   S706_ELE.Visu_Adv := W#16#300;
   S706_ELE.Visu_Ret := W#16#0;
   S706_ELE.Error_T1.IN := FALSE;
   S706_ELE.Error_T1.PT := T#7S;
   S706_ELE.Error_T1.Q := FALSE;
   S706_ELE.Error_T1.ET := T#0MS;
   S706_ELE.Error_T1.STATE := B#16#0;
   S706_ELE.Error_T1.STIME := T#23D5H8M52S101MS;
   S706_ELE.Error_T1.ATIME := T#23D5H8M52S353MS;
   S706_ELE.Error_T2.IN := FALSE;
   S706_ELE.Error_T2.PT := T#7S;
   S706_ELE.Error_T2.Q := FALSE;
   S706_ELE.Error_T2.ET := T#0MS;
   S706_ELE.Error_T2.STATE := B#16#0;
   S706_ELE.Error_T2.STIME := T#0MS;
   S706_ELE.Error_T2.ATIME := T#0MS;
   S706_ELE.CHK_Aux1 := FALSE;
   S706_ELE.CHK_Aux2 := FALSE;
   S706_ELE.Error_T1_DN := FALSE;
   S706_ELE.Error_T2_DN := FALSE;
   S706_ELE.Adv_Memo := TRUE;
   S706_ELE.Visu_Adv_Arr[0] := TRUE;
   S706_ELE.Visu_Adv_Arr[1] := TRUE;
   S706_ELE.Visu_Adv_Arr[2] := FALSE;
   S706_ELE.Visu_Adv_Arr[3] := FALSE;
   S706_ELE.Visu_Adv_Arr[4] := FALSE;
   S706_ELE.Visu_Adv_Arr[5] := FALSE;
   S706_ELE.Visu_Adv_Arr[6] := FALSE;
   S706_ELE.Visu_Adv_Arr[7] := FALSE;
   S706_ELE.Visu_Adv_Arr[8] := FALSE;
   S706_ELE.Visu_Adv_Arr[9] := FALSE;
   S706_ELE.Visu_Adv_Arr[10] := FALSE;
   S706_ELE.Visu_Adv_Arr[11] := FALSE;
   S706_ELE.Visu_Adv_Arr[12] := FALSE;
   S706_ELE.Visu_Adv_Arr[13] := FALSE;
   S706_ELE.Visu_Adv_Arr[14] := FALSE;
   S706_ELE.Visu_Adv_Arr[15] := FALSE;
   S706_ELE.Visu_Ret_Arr[0] := FALSE;
   S706_ELE.Visu_Ret_Arr[1] := FALSE;
   S706_ELE.Visu_Ret_Arr[2] := FALSE;
   S706_ELE.Visu_Ret_Arr[3] := FALSE;
   S706_ELE.Visu_Ret_Arr[4] := FALSE;
   S706_ELE.Visu_Ret_Arr[5] := FALSE;
   S706_ELE.Visu_Ret_Arr[6] := FALSE;
   S706_ELE.Visu_Ret_Arr[7] := FALSE;
   S706_ELE.Visu_Ret_Arr[8] := FALSE;
   S706_ELE.Visu_Ret_Arr[9] := FALSE;
   S706_ELE.Visu_Ret_Arr[10] := FALSE;
   S706_ELE.Visu_Ret_Arr[11] := FALSE;
   S706_ELE.Visu_Ret_Arr[12] := FALSE;
   S706_ELE.Visu_Ret_Arr[13] := FALSE;
   S706_ELE.Visu_Ret_Arr[14] := FALSE;
   S706_ELE.Visu_Ret_Arr[15] := FALSE;
   S706_ELE.BLK_Move_Ret := 0;
   S706_ELE.Enable := TRUE;
   S706_ELE.Adv_End := TRUE;
   S706_ELE.Ret_End := FALSE;
   S706_AIR_ELE.Enable_Aux := TRUE;
   S706_AIR_ELE.Adv_Amount := 1;
   S706_AIR_ELE.Ret_Amount := 1;
   S706_AIR_ELE.LS_Adv1 := TRUE;
   S706_AIR_ELE.LS_Ret1 := FALSE;
   S706_AIR_ELE.LS_Adv2 := FALSE;
   S706_AIR_ELE.LS_Ret2 := FALSE;
   S706_AIR_ELE.LS_Adv3 := FALSE;
   S706_AIR_ELE.LS_Ret3 := FALSE;
   S706_AIR_ELE.LS_Adv4 := FALSE;
   S706_AIR_ELE.LS_Ret4 := FALSE;
   S706_AIR_ELE.SOL_Adv := FALSE;
   S706_AIR_ELE.SOL_Ret := FALSE;
   S706_AIR_ELE.M_Ready := TRUE;
   S706_AIR_ELE.T_CHK1 := T#4S;
   S706_AIR_ELE.T_CHK2 := T#4S;
   S706_AIR_ELE.PB_Lamp_CHK := FALSE;
   S706_AIR_ELE.PB_Error_Rst := FALSE;
   S706_AIR_ELE.M_FLICK := TRUE;
   S706_AIR_ELE.M_Adv_Err := FALSE;
   S706_AIR_ELE.M_Ret_Err := FALSE;
   S706_AIR_ELE.LP_Adv := TRUE;
   S706_AIR_ELE.LP_Ret := FALSE;
   S706_AIR_ELE.Visu_Adv := W#16#300;
   S706_AIR_ELE.Visu_Ret := W#16#0;
   S706_AIR_ELE.Error_T1.IN := FALSE;
   S706_AIR_ELE.Error_T1.PT := T#4S;
   S706_AIR_ELE.Error_T1.Q := FALSE;
   S706_AIR_ELE.Error_T1.ET := T#0MS;
   S706_AIR_ELE.Error_T1.STATE := B#16#0;
   S706_AIR_ELE.Error_T1.STIME := T#23D5H8M44S377MS;
   S706_AIR_ELE.Error_T1.ATIME := T#23D5H8M44S470MS;
   S706_AIR_ELE.Error_T2.IN := FALSE;
   S706_AIR_ELE.Error_T2.PT := T#4S;
   S706_AIR_ELE.Error_T2.Q := FALSE;
   S706_AIR_ELE.Error_T2.ET := T#0MS;
   S706_AIR_ELE.Error_T2.STATE := B#16#0;
   S706_AIR_ELE.Error_T2.STIME := T#0MS;
   S706_AIR_ELE.Error_T2.ATIME := T#0MS;
   S706_AIR_ELE.CHK_Aux1 := FALSE;
   S706_AIR_ELE.CHK_Aux2 := FALSE;
   S706_AIR_ELE.Error_T1_DN := FALSE;
   S706_AIR_ELE.Error_T2_DN := FALSE;
   S706_AIR_ELE.Adv_Memo := TRUE;
   S706_AIR_ELE.Visu_Adv_Arr[0] := TRUE;
   S706_AIR_ELE.Visu_Adv_Arr[1] := TRUE;
   S706_AIR_ELE.Visu_Adv_Arr[2] := FALSE;
   S706_AIR_ELE.Visu_Adv_Arr[3] := FALSE;
   S706_AIR_ELE.Visu_Adv_Arr[4] := FALSE;
   S706_AIR_ELE.Visu_Adv_Arr[5] := FALSE;
   S706_AIR_ELE.Visu_Adv_Arr[6] := FALSE;
   S706_AIR_ELE.Visu_Adv_Arr[7] := FALSE;
   S706_AIR_ELE.Visu_Adv_Arr[8] := FALSE;
   S706_AIR_ELE.Visu_Adv_Arr[9] := FALSE;
   S706_AIR_ELE.Visu_Adv_Arr[10] := FALSE;
   S706_AIR_ELE.Visu_Adv_Arr[11] := FALSE;
   S706_AIR_ELE.Visu_Adv_Arr[12] := FALSE;
   S706_AIR_ELE.Visu_Adv_Arr[13] := FALSE;
   S706_AIR_ELE.Visu_Adv_Arr[14] := FALSE;
   S706_AIR_ELE.Visu_Adv_Arr[15] := FALSE;
   S706_AIR_ELE.Visu_Ret_Arr[0] := FALSE;
   S706_AIR_ELE.Visu_Ret_Arr[1] := FALSE;
   S706_AIR_ELE.Visu_Ret_Arr[2] := FALSE;
   S706_AIR_ELE.Visu_Ret_Arr[3] := FALSE;
   S706_AIR_ELE.Visu_Ret_Arr[4] := FALSE;
   S706_AIR_ELE.Visu_Ret_Arr[5] := FALSE;
   S706_AIR_ELE.Visu_Ret_Arr[6] := FALSE;
   S706_AIR_ELE.Visu_Ret_Arr[7] := FALSE;
   S706_AIR_ELE.Visu_Ret_Arr[8] := FALSE;
   S706_AIR_ELE.Visu_Ret_Arr[9] := FALSE;
   S706_AIR_ELE.Visu_Ret_Arr[10] := FALSE;
   S706_AIR_ELE.Visu_Ret_Arr[11] := FALSE;
   S706_AIR_ELE.Visu_Ret_Arr[12] := FALSE;
   S706_AIR_ELE.Visu_Ret_Arr[13] := FALSE;
   S706_AIR_ELE.Visu_Ret_Arr[14] := FALSE;
   S706_AIR_ELE.Visu_Ret_Arr[15] := FALSE;
   S706_AIR_ELE.BLK_Move_Ret := 0;
   S706_AIR_ELE.Enable := TRUE;
   S706_AIR_ELE.Adv_End := TRUE;
   S706_AIR_ELE.Ret_End := FALSE;
END_DATA_BLOCK

FUNCTION FC 121 : VOID
TITLE =
VERSION : 0.1

BEGIN
NETWORK
TITLE =
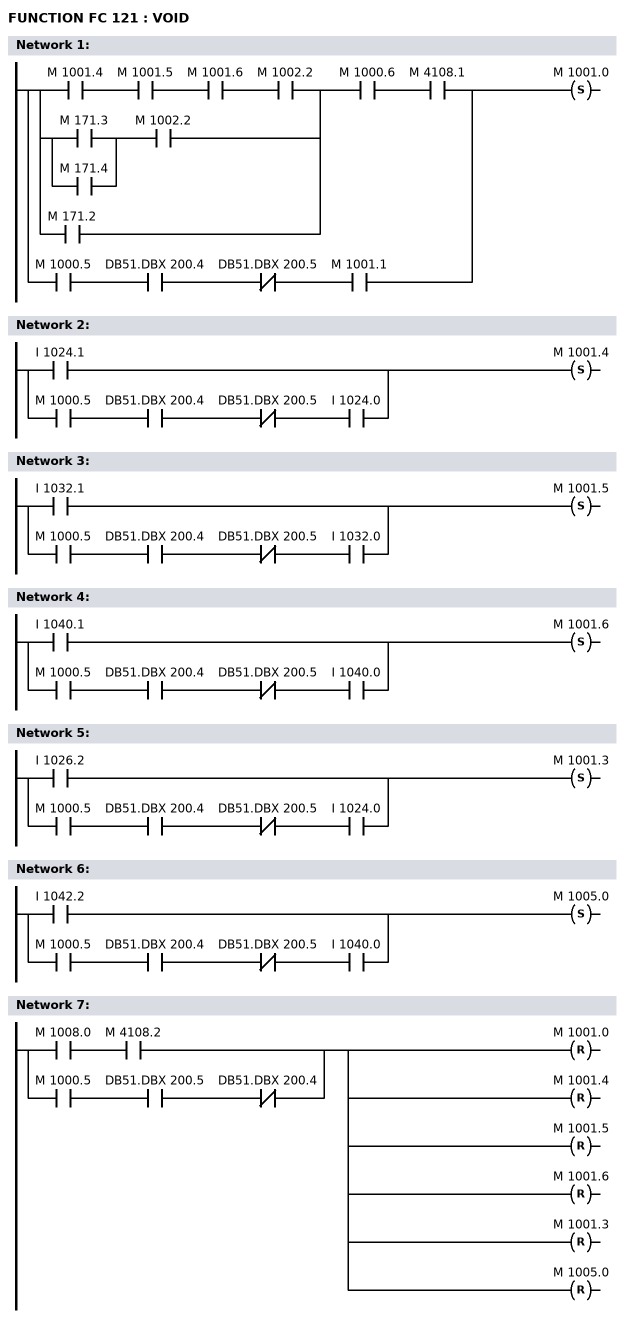

      A(    ;
      A     M   1001.4;
      A     M   1001.5;
      A     M   1001.6;
      A     M   1002.2;
      O     ;
      A(    ;
      O     M    171.3;
      O     M    171.4;
      )     ;
      A     M   1002.2;
      O     M    171.2;
      )     ;
      A     M   1000.6;
      A     M   4108.1;
      O     ;
      A     M   1000.5;
      A     DB51.DBX  200.4;
      AN    DB51.DBX  200.5;
      A     M   1001.1;
      S     M   1001.0;
NETWORK
TITLE =

      O     I   1024.1;
      O     ;
      A     M   1000.5;
      A     DB51.DBX  200.4;
      AN    DB51.DBX  200.5;
      A     I   1024.0;
      S     M   1001.4;
NETWORK
TITLE =

      O     I   1032.1;
      O     ;
      A     M   1000.5;
      A     DB51.DBX  200.4;
      AN    DB51.DBX  200.5;
      A     I   1032.0;
      S     M   1001.5;
NETWORK
TITLE =

      O     I   1040.1;
      O     ;
      A     M   1000.5;
      A     DB51.DBX  200.4;
      AN    DB51.DBX  200.5;
      A     I   1040.0;
      S     M   1001.6;
NETWORK
TITLE =

      O     I   1026.2;
      O     ;
      A     M   1000.5;
      A     DB51.DBX  200.4;
      AN    DB51.DBX  200.5;
      A     I   1024.0;
      S     M   1001.3;
NETWORK
TITLE =

      O     I   1042.2;
      O     ;
      A     M   1000.5;
      A     DB51.DBX  200.4;
      AN    DB51.DBX  200.5;
      A     I   1040.0;
      S     M   1005.0;
NETWORK
TITLE =

      A     M   1008.0;
      A     M   4108.2;
      O     ;
      A     M   1000.5;
      A     DB51.DBX  200.5;
      AN    DB51.DBX  200.4;
      R     M   1001.0;
      R     M   1001.4;
      R     M   1001.5;
      R     M   1001.6;
      R     M   1001.3;
      R     M   1005.0;
END_FUNCTION

FUNCTION_BLOCK FB 122
TITLE =
VERSION : 0.1

BEGIN
NETWORK
TITLE =
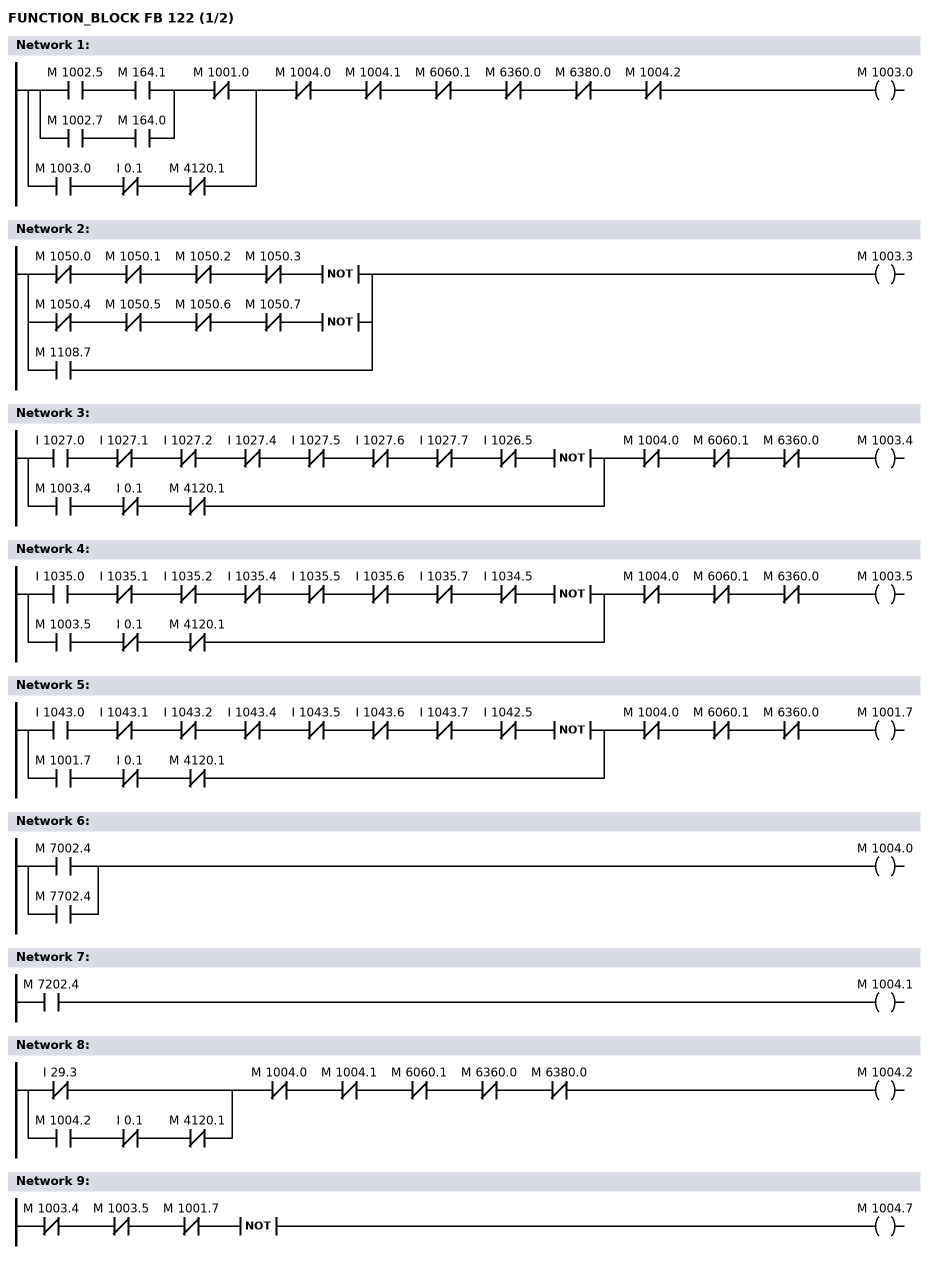

      A(    ;
      A(    ;
      A     M   1002.5;
      A     M    164.1;
      O     ;
      A     M   1002.7;
      A     M    164.0;
      )     ;
      AN    M   1001.0;
      O     ;
      A     M   1003.0;
      AN    I      0.1;
      AN    M   4120.1;
      )     ;
      AN    M   1004.0;
      AN    M   1004.1;
      AN    M   6060.1;
      AN    M   6360.0;
      AN    M   6380.0;
      AN    M   1004.2;
      =     M   1003.0;
NETWORK
TITLE =

      AN    M   1050.0;
      AN    M   1050.1;
      AN    M   1050.2;
      AN    M   1050.3;
      NOT   ;
      O(    ;
      AN    M   1050.4;
      AN    M   1050.5;
      AN    M   1050.6;
      AN    M   1050.7;
      NOT   ;
      )     ;
      O     M   1108.7;
      =     M   1003.3;
NETWORK
TITLE =

      A(    ;
      A     I   1027.0;
      AN    I   1027.1;
      AN    I   1027.2;
      AN    I   1027.4;
      AN    I   1027.5;
      AN    I   1027.6;
      AN    I   1027.7;
      AN    I   1026.5;
      NOT   ;
      O     ;
      A     M   1003.4;
      AN    I      0.1;
      AN    M   4120.1;
      )     ;
      AN    M   1004.0;
      AN    M   6060.1;
      AN    M   6360.0;
      =     M   1003.4;
NETWORK
TITLE =

      A(    ;
      A     I   1035.0;
      AN    I   1035.1;
      AN    I   1035.2;
      AN    I   1035.4;
      AN    I   1035.5;
      AN    I   1035.6;
      AN    I   1035.7;
      AN    I   1034.5;
      NOT   ;
      O     ;
      A     M   1003.5;
      AN    I      0.1;
      AN    M   4120.1;
      )     ;
      AN    M   1004.0;
      AN    M   6060.1;
      AN    M   6360.0;
      =     M   1003.5;
NETWORK
TITLE =

      A(    ;
      A     I   1043.0;
      AN    I   1043.1;
      AN    I   1043.2;
      AN    I   1043.4;
      AN    I   1043.5;
      AN    I   1043.6;
      AN    I   1043.7;
      AN    I   1042.5;
      NOT   ;
      O     ;
      A     M   1001.7;
      AN    I      0.1;
      AN    M   4120.1;
      )     ;
      AN    M   1004.0;
      AN    M   6060.1;
      AN    M   6360.0;
      =     M   1001.7;
NETWORK
TITLE =

      O     M   7002.4;
      O     M   7702.4;
      =     M   1004.0;
NETWORK
TITLE =

      A     M   7202.4;
      =     M   1004.1;
NETWORK
TITLE =

      A(    ;
      ON    I     29.3;
      O     ;
      A     M   1004.2;
      AN    I      0.1;
      AN    M   4120.1;
      )     ;
      AN    M   1004.0;
      AN    M   1004.1;
      AN    M   6060.1;
      AN    M   6360.0;
      AN    M   6380.0;
      =     M   1004.2;
NETWORK
TITLE =

      AN    M   1003.4;
      AN    M   1003.5;
      AN    M   1001.7;
      NOT   ;
      =     M   1004.7;
NETWORK
TITLE =
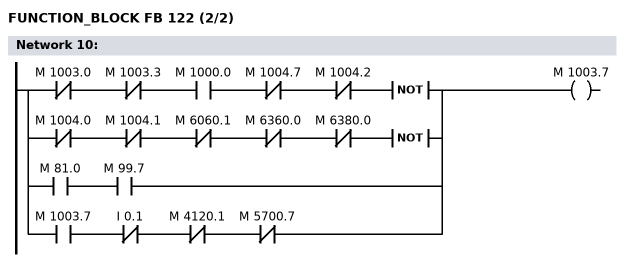

      AN    M   1003.0;
      AN    M   1003.3;
      A     M   1000.0;
      AN    M   1004.7;
      AN    M   1004.2;
      NOT   ;
      O(    ;
      AN    M   1004.0;
      AN    M   1004.1;
      AN    M   6060.1;
      AN    M   6360.0;
      AN    M   6380.0;
      NOT   ;
      )     ;
      O     ;
      A     M     81.0;
      A     M     99.7;
      O     ;
      A     M   1003.7;
      AN    I      0.1;
      AN    M   4120.1;
      AN    M   5700.7;
      =     M   1003.7;
END_FUNCTION_BLOCK

DATA_BLOCK DB 122
TITLE =
VERSION : 0.0

 FB 122
BEGIN
END_DATA_BLOCK

FUNCTION FC 122 : VOID
TITLE =
VERSION : 0.1

BEGIN
NETWORK
TITLE =
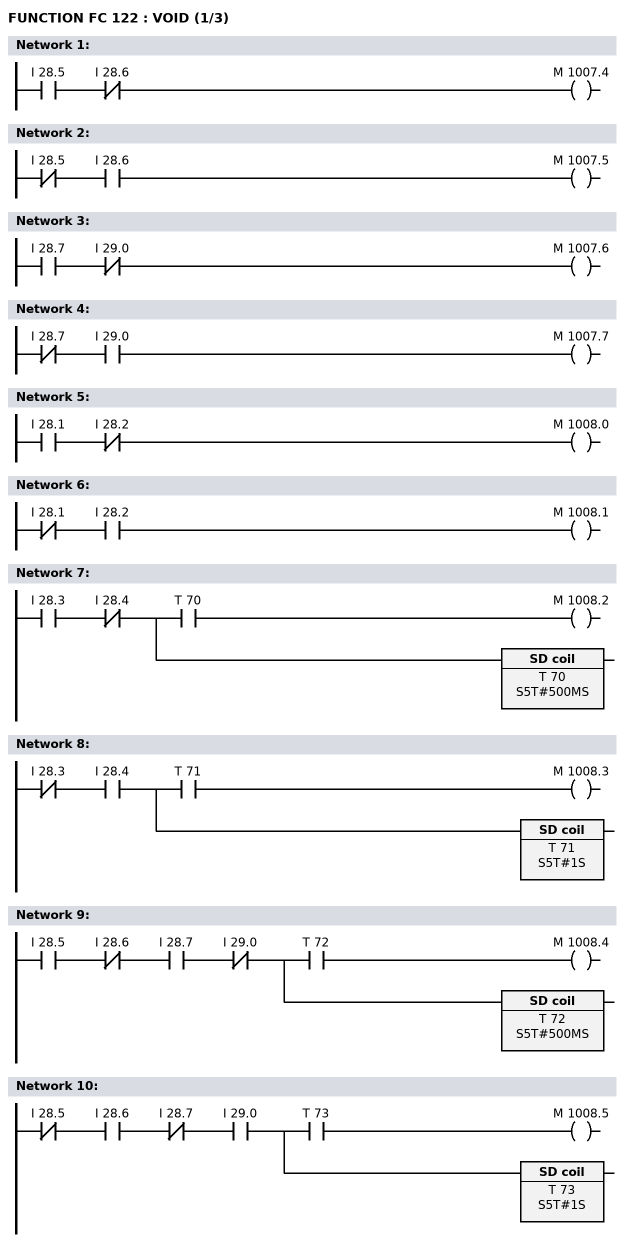

      A     I     28.5;
      AN    I     28.6;
      =     M   1007.4;
NETWORK
TITLE =

      AN    I     28.5;
      A     I     28.6;
      =     M   1007.5;
NETWORK
TITLE =

      A     I     28.7;
      AN    I     29.0;
      =     M   1007.6;
NETWORK
TITLE =

      AN    I     28.7;
      A     I     29.0;
      =     M   1007.7;
NETWORK
TITLE =

      A     I     28.1;
      AN    I     28.2;
      =     M   1008.0;
NETWORK
TITLE =

      AN    I     28.1;
      A     I     28.2;
      =     M   1008.1;
NETWORK
TITLE =

      A     I     28.3;
      AN    I     28.4;
      =     L      0.0;
      A     L      0.0;
      A     T     70;
      =     M   1008.2;
      A     L      0.0;
      BLD   102;
      L     S5T#500MS;
      SD    T     70;
NETWORK
TITLE =

      AN    I     28.3;
      A     I     28.4;
      =     L      0.0;
      A     L      0.0;
      A     T     71;
      =     M   1008.3;
      A     L      0.0;
      BLD   102;
      L     S5T#1S;
      SD    T     71;
NETWORK
TITLE =

      A     I     28.5;
      AN    I     28.6;
      A     I     28.7;
      AN    I     29.0;
      =     L      0.0;
      A     L      0.0;
      A     T     72;
      =     M   1008.4;
      A     L      0.0;
      BLD   102;
      L     S5T#500MS;
      SD    T     72;
NETWORK
TITLE =

      AN    I     28.5;
      A     I     28.6;
      AN    I     28.7;
      A     I     29.0;
      =     L      0.0;
      A     L      0.0;
      A     T     73;
      =     M   1008.5;
      A     L      0.0;
      BLD   102;
      L     S5T#1S;
      SD    T     73;
NETWORK
TITLE =#706 급전POWER전원
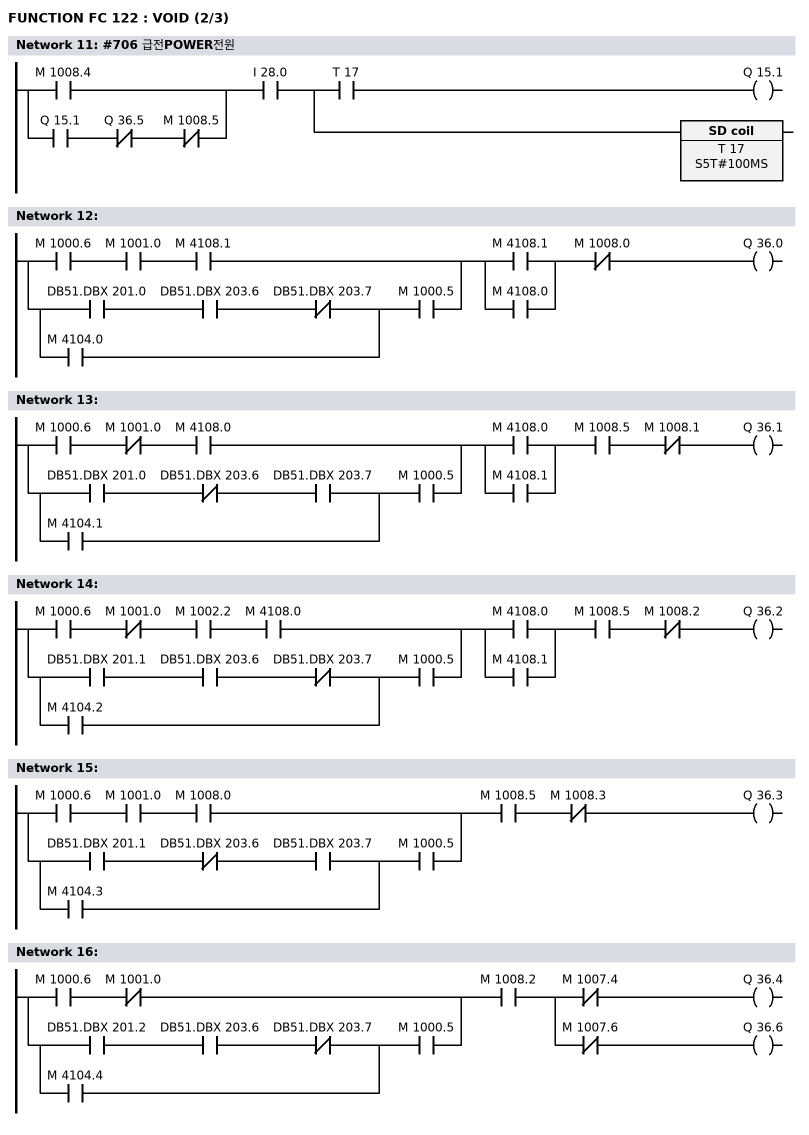

      A(    ;
      O     M   1008.4;
      O     ;
      A     Q     15.1;
      AN    Q     36.5;
      AN    M   1008.5;
      )     ;
      A     I     28.0;
      =     L      0.0;
      A     L      0.0;
      A     T     17;
      =     Q     15.1;
      A     L      0.0;
      BLD   102;
      L     S5T#100MS;
      SD    T     17;
NETWORK
TITLE =

      A(    ;
      A     M   1000.6;
      A     M   1001.0;
      A     M   4108.1;
      O     ;
      A(    ;
      A     DB51.DBX  201.0;
      A     DB51.DBX  203.6;
      AN    DB51.DBX  203.7;
      O     M   4104.0;
      )     ;
      A     M   1000.5;
      )     ;
      A(    ;
      O     M   4108.1;
      O     M   4108.0;
      )     ;
      AN    M   1008.0;
      =     Q     36.0;
NETWORK
TITLE =

      A(    ;
      A     M   1000.6;
      AN    M   1001.0;
      A     M   4108.0;
      O     ;
      A(    ;
      A     DB51.DBX  201.0;
      AN    DB51.DBX  203.6;
      A     DB51.DBX  203.7;
      O     M   4104.1;
      )     ;
      A     M   1000.5;
      )     ;
      A(    ;
      O     M   4108.0;
      O     M   4108.1;
      )     ;
      A     M   1008.5;
      AN    M   1008.1;
      =     Q     36.1;
NETWORK
TITLE =

      A(    ;
      A     M   1000.6;
      AN    M   1001.0;
      A     M   1002.2;
      A     M   4108.0;
      O     ;
      A(    ;
      A     DB51.DBX  201.1;
      A     DB51.DBX  203.6;
      AN    DB51.DBX  203.7;
      O     M   4104.2;
      )     ;
      A     M   1000.5;
      )     ;
      A(    ;
      O     M   4108.0;
      O     M   4108.1;
      )     ;
      A     M   1008.5;
      AN    M   1008.2;
      =     Q     36.2;
NETWORK
TITLE =

      A(    ;
      A     M   1000.6;
      A     M   1001.0;
      A     M   1008.0;
      O     ;
      A(    ;
      A     DB51.DBX  201.1;
      AN    DB51.DBX  203.6;
      A     DB51.DBX  203.7;
      O     M   4104.3;
      )     ;
      A     M   1000.5;
      )     ;
      A     M   1008.5;
      AN    M   1008.3;
      =     Q     36.3;
NETWORK
TITLE =

      A(    ;
      A     M   1000.6;
      AN    M   1001.0;
      O     ;
      A(    ;
      A     DB51.DBX  201.2;
      A     DB51.DBX  203.6;
      AN    DB51.DBX  203.7;
      O     M   4104.4;
      )     ;
      A     M   1000.5;
      )     ;
      A     M   1008.2;
      =     L      0.0;
      A     L      0.0;
      AN    M   1007.4;
      =     Q     36.4;
      A     L      0.0;
      AN    M   1007.6;
      =     Q     36.6;
NETWORK
TITLE =
